LIN {X 0,Y 238.597,Z 271.892,A -85,B 0,C 180,E1 -19740.745,E2 -19740.745} C_VEL
LIN {X 0,Y 234.921,Z 263.135,A -85,B 0,C 180,E1 -19741.833,E2 -19741.833} C_VEL
LIN {X 0,Y 234.766,Z 262.386,A -85,B 0,C 180,E1 -19741.948,E2 -19741.948} C_VEL
LIN {X 0,Y 234.827,Z 259.801,A -85,B 0,C 180,E1 -19746.092,E2 -19746.092} C_VEL
LIN {X 0,Y 234.795,Z 259.401,A -85,B 0,C 180,E1 -19746.773,E2 -19746.773} C_VEL
LIN {X 0,Y 234.887,Z 259.23,A -85,B 0,C 180,E1 -19748.927,E2 -19748.927} C_VEL
LIN {X 0,Y 234.889,Z 259.225,A -85,B 0,C 180,E1 -19753.486,E2 -19753.486} C_VEL
LIN {X 0,Y 234.888,Z 259.222,A -85,B 0,C 180,E1 -19756.514,E2 -19756.514} C_VEL
LIN {X 0,Y 234.92,Z 259.222,A -85,B 0,C 180,E1 -19761.079,E2 -19761.079} C_VEL
LIN {X 0,Y 234.932,Z 259.222,A -85,B 0,C 180,E1 -19765.362,E2 -19765.362} C_VEL
LIN {X 0,Y 234.9,Z 259.224,A -85,B 0,C 180,E1 -19769.427,E2 -19769.427} C_VEL
LIN {X 0,Y 234.97,Z 259.215,A -85,B 0,C 180,E1 -19773.806,E2 -19773.806} C_VEL
LIN {X 0,Y 234.99,Z 259.212,A -85,B 0,C 180,E1 -19778.968,E2 -19778.968} C_VEL
LIN {X 0,Y 235.057,Z 259.206,A -85,B 0,C 180,E1 -19783.092,E2 -19783.092} C_VEL
LIN {X 0,Y 235.116,Z 259.196,A -85,B 0,C 180,E1 -19787.922,E2 -19787.922} C_VEL
LIN {X 0,Y 235.392,Z 259.162,A -85,B 0,C 180,E1 -19791.415,E2 -19791.415} C_VEL
LIN {X 0,Y 235.406,Z 259.16,A -85,B 0,C 180,E1 -19793.141,E2 -19793.141} C_VEL
LIN {X 0,Y 235.582,Z 259.141,A -85,B 0,C 180,E1 -19798.29,E2 -19798.29} C_VEL
LIN {X 0,Y 235.597,Z 259.138,A -85,B 0,C 180,E1 -19801.709,E2 -19801.709} C_VEL
LIN {X 0,Y 235.37,Z 259.165,A -85,B 0,C 180,E1 -19806.86,E2 -19806.86} C_VEL
LIN {X 0,Y 235.216,Z 259.185,A -85,B 0,C 180,E1 -19810.327,E2 -19810.327} C_VEL
LIN {X 0,Y 235.116,Z 259.195,A -85,B 0,C 180,E1 -19815.606,E2 -19815.606} C_VEL
LIN {X 0,Y 235.005,Z 259.212,A -85,B 0,C 180,E1 -19819.206,E2 -19819.206} C_VEL
LIN {X 0,Y 234.927,Z 259.223,A -85,B 0,C 180,E1 -19822.886,E2 -19822.886} C_VEL
LIN {X 0,Y 234.927,Z 259.226,A -85,B 0,C 180,E1 -19826.663,E2 -19826.663} C_VEL
LIN {X 0,Y 234.937,Z 259.227,A -85,B 0,C 180,E1 -19831.568,E2 -19831.568} C_VEL
LIN {X 0,Y 234.987,Z 259.521,A -85,B 0,C 180,E1 -19832.571,E2 -19832.571} C_VEL
LIN {X 0,Y 235.549,Z 262.75,A -85,B 0,C 180,E1 -19836.636,E2 -19836.636} C_VEL
LIN {X 0,Y 236.203,Z 266.509,A -85,B 0,C 180,E1 -19840.889,E2 -19840.889} C_VEL
LIN {X 0,Y 237.07,Z 270.768,A -85,B 0,C 180,E1 -19845.356,E2 -19845.356} C_VEL
LIN {X 0,Y 237.855,Z 274.98,A -85,B 0,C 180,E1 -19849.455,E2 -19849.455} C_VEL
LIN {X 0,Y 237.937,Z 275.641,A -85,B 0,C 180,E1 -19850.071,E2 -19850.071} C_VEL
LIN {X 0,Y 237.706,Z 276.681,A -85,B 0,C 180,E1 -19850.982,E2 -19850.982} C_VEL
LIN {X 0,Y 236.882,Z 277.795,A -85,B 0,C 180,E1 -19851.872,E2 -19851.872} C_VEL
LIN {X 0,Y 234.22,Z 280.117,A -85,B 0,C 180,E1 -19853.609,E2 -19853.609} C_VEL
LIN {X 0,Y 231.328,Z 282.486,A -85,B 0,C 180,E1 -19855.381,E2 -19855.381} C_VEL
LIN {X 0,Y 229.905,Z 284.219,A -85,B 0,C 180,E1 -19856.776,E2 -19856.776} C_VEL
LIN {X 0,Y 229.7,Z 284.777,A -85,B 0,C 180,E1 -19857.256,E2 -19857.256} C_VEL
LIN {X 0,Y 233.573,Z 300.662,A -85,B 0,C 180,E1 -19858.908,E2 -19858.908} C_VEL
LIN {X 0,Y 235.544,Z 312.113,A -85,B 0,C 180,E1 -19860.268,E2 -19860.268} C_VEL
LIN {X 0,Y 236.725,Z 323.693,A -85,B 0,C 180,E1 -19861.844,E2 -19861.844} C_VEL
LIN {X 0,Y 237.034,Z 334.803,A -85,B 0,C 180,E1 -19863.593,E2 -19863.593} C_VEL
LIN {X 0,Y 236.7,Z 344.769,A -85,B 0,C 180,E1 -19865.438,E2 -19865.438} C_VEL
LIN {X 0,Y 234.724,Z 352.959,A -85,B 0,C 180,E1 -19867.093,E2 -19867.093} C_VEL
LIN {X 0,Y 232.482,Z 361.592,A -85,B 0,C 180,E1 -19869.232,E2 -19869.232} C_VEL
LIN {X 0,Y 230.493,Z 369.799,A -85,B 0,C 180,E1 -19871.788,E2 -19871.788} C_VEL
LIN {X 0,Y 228.678,Z 376.512,A -85,B 0,C 180,E1 -19874.4,E2 -19874.4} C_VEL
LIN {X 0,Y 227.13,Z 382.668,A -85,B 0,C 180,E1 -19877.491,E2 -19877.491} C_VEL
LIN {X 0,Y 226.362,Z 386.685,A -85,B 0,C 180,E1 -19880.168,E2 -19880.168} C_VEL
LIN {X 0,Y 225.939,Z 389.662,A -85,B 0,C 180,E1 -19882.853,E2 -19882.853} C_VEL
LIN {X 0,Y 225.845,Z 391.153,A -85,B 0,C 180,E1 -19884.748,E2 -19884.748} C_VEL
LIN {X 0,Y 225.843,Z 392.104,A -85,B 0,C 180,E1 -19886.432,E2 -19886.432} C_VEL
LIN {X 0,Y 225.89,Z 392.728,A -85,B 0,C 180,E1 -19888.217,E2 -19888.217} C_VEL
LIN {X 0,Y 225.95,Z 392.949,A -85,B 0,C 180,E1 -19890,E2 -19890} C_VEL
LIN {X 0,Y 225.89,Z 392.72,A -85,B 0,C 180,E1 -19891.783,E2 -19891.783} C_VEL
LIN {X 0,Y 225.839,Z 392.091,A -85,B 0,C 180,E1 -19893.569,E2 -19893.569} C_VEL
LIN {X 0,Y 225.842,Z 391.068,A -85,B 0,C 180,E1 -19895.357,E2 -19895.357} C_VEL
LIN {X 0,Y 225.937,Z 389.637,A -85,B 0,C 180,E1 -19897.148,E2 -19897.148} C_VEL
LIN {X 0,Y 226.357,Z 386.646,A -85,B 0,C 180,E1 -19899.833,E2 -19899.833} C_VEL
LIN {X 0,Y 227.131,Z 382.613,A -85,B 0,C 180,E1 -19902.51,E2 -19902.51} C_VEL
LIN {X 0,Y 228.676,Z 376.437,A -85,B 0,C 180,E1 -19905.6,E2 -19905.6} C_VEL
LIN {X 0,Y 230.502,Z 369.708,A -85,B 0,C 180,E1 -19908.212,E2 -19908.212} C_VEL
LIN {X 0,Y 232.694,Z 360.843,A -85,B 0,C 180,E1 -19910.942,E2 -19910.942} C_VEL
LIN {X 0,Y 234.721,Z 352.815,A -85,B 0,C 180,E1 -19912.908,E2 -19912.908} C_VEL
LIN {X 0,Y 236.682,Z 344.6,A -85,B 0,C 180,E1 -19914.565,E2 -19914.565} C_VEL
LIN {X 0,Y 236.994,Z 334.585,A -85,B 0,C 180,E1 -19916.412,E2 -19916.412} C_VEL
LIN {X 0,Y 236.678,Z 323.434,A -85,B 0,C 180,E1 -19918.158,E2 -19918.158} C_VEL
LIN {X 0,Y 235.469,Z 311.893,A -85,B 0,C 180,E1 -19919.725,E2 -19919.725} C_VEL
LIN {X 0,Y 233.198,Z 299.127,A -85,B 0,C 180,E1 -19921.229,E2 -19921.229} C_VEL
LIN {X 0,Y 230.268,Z 287.553,A -85,B 0,C 180,E1 -19922.422,E2 -19922.422} C_VEL
LIN {X 0,Y 229.666,Z 284.769,A -85,B 0,C 180,E1 -19922.666,E2 -19922.666} C_VEL
LIN {X 0,Y 230.806,Z 280.466,A -85,B 0,C 180,E1 -19926.426,E2 -19926.426} C_VEL
LIN {X 0,Y 231.021,Z 278.054,A -85,B 0,C 180,E1 -19928.629,E2 -19928.629} C_VEL
LIN {X 0,Y 230.853,Z 276.123,A -85,B 0,C 180,E1 -19930.439,E2 -19930.439} C_VEL
LIN {X 0,Y 230.037,Z 271.961,A -85,B 0,C 180,E1 -19934.644,E2 -19934.644} C_VEL
LIN {X 0,Y 229.522,Z 269.108,A -85,B 0,C 180,E1 -19937.651,E2 -19937.651} C_VEL
LIN {X 0,Y 228.67,Z 264.453,A -85,B 0,C 180,E1 -19943.044,E2 -19943.044} C_VEL
LIN {X 0,Y 228.208,Z 261.833,A -85,B 0,C 180,E1 -19946.335,E2 -19946.335} C_VEL
LIN {X 0,Y 227.893,Z 260.097,A -85,B 0,C 180,E1 -19948.761,E2 -19948.761} C_VEL
LIN {X 0,Y 227.906,Z 260.098,A -85,B 0,C 180,E1 -19953.418,E2 -19953.418} C_VEL
LIN {X 0,Y 227.95,Z 260.093,A -85,B 0,C 180,E1 -19958.286,E2 -19958.286} C_VEL
LIN {X 0,Y 228.037,Z 260.08,A -85,B 0,C 180,E1 -19962.827,E2 -19962.827} C_VEL
LIN {X 0,Y 228.075,Z 260.076,A -85,B 0,C 180,E1 -19967.543,E2 -19967.543} C_VEL
LIN {X 0,Y 228.266,Z 260.051,A -85,B 0,C 180,E1 -19971.145,E2 -19971.145} C_VEL
LIN {X 0,Y 228.321,Z 260.043,A -85,B 0,C 180,E1 -19972.928,E2 -19972.928} C_VEL
LIN {X 0,Y 228.558,Z 260.014,A -85,B 0,C 180,E1 -19978.238,E2 -19978.238} C_VEL
LIN {X 0,Y 228.542,Z 260.018,A -85,B 0,C 180,E1 -19981.762,E2 -19981.762} C_VEL
LIN {X 0,Y 228.319,Z 260.044,A -85,B 0,C 180,E1 -19987.073,E2 -19987.073} C_VEL
LIN {X 0,Y 228.146,Z 260.066,A -85,B 0,C 180,E1 -19990.651,E2 -19990.651} C_VEL
LIN {X 0,Y 228.041,Z 260.078,A -85,B 0,C 180,E1 -19994.274,E2 -19994.274} C_VEL
LIN {X 0,Y 227.957,Z 260.086,A -85,B 0,C 180,E1 -19997.957,E2 -19997.957} C_VEL
LIN {X 0,Y 227.923,Z 260.094,A -85,B 0,C 180,E1 -20002.323,E2 -20002.323} C_VEL
LIN {X 0,Y 227.925,Z 260.094,A -85,B 0,C 180,E1 -20006.592,E2 -20006.592} C_VEL
LIN {X 0,Y 227.876,Z 260.101,A -85,B 0,C 180,E1 -20010.281,E2 -20010.281} C_VEL
LIN {X 0,Y 227.88,Z 260.098,A -85,B 0,C 180,E1 -20013.72,E2 -20013.72} C_VEL
LIN {X 0,Y 227.847,Z 260.105,A -85,B 0,C 180,E1 -20018.091,E2 -20018.091} C_VEL
LIN {X 0,Y 227.814,Z 260.106,A -85,B 0,C 180,E1 -20022.742,E2 -20022.742} C_VEL
LIN {X 0,Y 227.811,Z 260.106,A -85,B 0,C 180,E1 -20027.257,E2 -20027.257} C_VEL
LIN {X 0,Y 227.816,Z 260.107,A -85,B 0,C 180,E1 -20030.465,E2 -20030.465} C_VEL
LIN {X 0,Y 227.783,Z 260.111,A -85,B 0,C 180,E1 -20031.896,E2 -20031.896} C_VEL
LIN {X 0,Y 227.833,Z 261.048,A -85,B 0,C 180,E1 -20034.119,E2 -20034.119} C_VEL
LIN {X 0,Y 227.804,Z 262.883,A -85,B 0,C 180,E1 -20037.124,E2 -20037.124} C_VEL
LIN {X 0,Y 228.901,Z 265.947,A -85,B 0,C 180,E1 -20037.508,E2 -20037.508} C_VEL
LIN {X 0,Y 233.368,Z 276.685,A -85,B 0,C 180,E1 -20038.978,E2 -20038.978} C_VEL
LIN {X 0,Y 236.842,Z 287.16,A -85,B 0,C 180,E1 -20040.513,E2 -20040.513} C_VEL
LIN {X 0,Y 239.401,Z 297.64,A -85,B 0,C 180,E1 -20042.174,E2 -20042.174} C_VEL
LIN {X 0,Y 240.91,Z 306.572,A -85,B 0,C 180,E1 -20043.735,E2 -20043.735} C_VEL
LIN {X 0,Y 241.071,Z 308.452,A -85,B 0,C 180,E1 -20044.068,E2 -20044.068} C_VEL
LIN {X 0,Y 239.057,Z 318.286,A -85,B 0,C 180,E1 -20045.695,E2 -20045.695} C_VEL
LIN {X 0,Y 236.799,Z 328.203,A -85,B 0,C 180,E1 -20047.764,E2 -20047.764} C_VEL
LIN {X 0,Y 234.201,Z 337.802,A -85,B 0,C 180,E1 -20050.269,E2 -20050.269} C_VEL
LIN {X 0,Y 231.99,Z 345.446,A -85,B 0,C 180,E1 -20052.82,E2 -20052.82} C_VEL
LIN {X 0,Y 230.501,Z 350.658,A -85,B 0,C 180,E1 -20054.979,E2 -20054.979} C_VEL
LIN {X 0,Y 228.915,Z 355.716,A -85,B 0,C 180,E1 -20057.589,E2 -20057.589} C_VEL
LIN {X 0,Y 227.809,Z 359.633,A -85,B 0,C 180,E1 -20060.231,E2 -20060.231} C_VEL
LIN {X 0,Y 227.03,Z 362.522,A -85,B 0,C 180,E1 -20062.887,E2 -20062.887} C_VEL
LIN {X 0,Y 226.641,Z 363.904,A -85,B 0,C 180,E1 -20064.662,E2 -20064.662} C_VEL
LIN {X 0,Y 226.13,Z 365.496,A -85,B 0,C 180,E1 -20068.219,E2 -20068.219} C_VEL
LIN {X 0,Y 226.084,Z 365.723,A -85,B 0,C 180,E1 -20070,E2 -20070} C_VEL
LIN {X 0,Y 226.313,Z 364.946,A -85,B 0,C 180,E1 -20073.561,E2 -20073.561} C_VEL
LIN {X 0,Y 226.627,Z 363.983,A -85,B 0,C 180,E1 -20075.338,E2 -20075.338} C_VEL
LIN {X 0,Y 227.3,Z 361.44,A -85,B 0,C 180,E1 -20078.339,E2 -20078.339} C_VEL
LIN {X 0,Y 228.481,Z 357.329,A -85,B 0,C 180,E1 -20081.533,E2 -20081.533} C_VEL
LIN {X 0,Y 229.836,Z 352.722,A -85,B 0,C 180,E1 -20084.16,E2 -20084.16} C_VEL
LIN {X 0,Y 231.915,Z 345.77,A -85,B 0,C 180,E1 -20087.185,E2 -20087.185} C_VEL
LIN {X 0,Y 234.129,Z 338.223,A -85,B 0,C 180,E1 -20089.737,E2 -20089.737} C_VEL
LIN {X 0,Y 236.736,Z 328.716,A -85,B 0,C 180,E1 -20092.241,E2 -20092.241} C_VEL
LIN {X 0,Y 238.959,Z 318.91,A -85,B 0,C 180,E1 -20094.315,E2 -20094.315} C_VEL
LIN {X 0,Y 241.151,Z 308.24,A -85,B 0,C 180,E1 -20096.091,E2 -20096.091} C_VEL
LIN {X 0,Y 239.528,Z 298.088,A -85,B 0,C 180,E1 -20097.884,E2 -20097.884} C_VEL
LIN {X 0,Y 237.21,Z 288.374,A -85,B 0,C 180,E1 -20099.441,E2 -20099.441} C_VEL
LIN {X 0,Y 233.811,Z 277.855,A -85,B 0,C 180,E1 -20100.998,E2 -20100.998} C_VEL
LIN {X 0,Y 229.349,Z 266.623,A -85,B 0,C 180,E1 -20102.523,E2 -20102.523} C_VEL
LIN {X 0,Y 227.97,Z 263.675,A -85,B 0,C 180,E1 -20102.921,E2 -20102.921} C_VEL
LIN {X 0,Y 227.812,Z 262.875,A -85,B 0,C 180,E1 -20103.011,E2 -20103.011} C_VEL
LIN {X 0,Y 227.807,Z 260.688,A -85,B 0,C 180,E1 -20106.667,E2 -20106.667} C_VEL
LIN {X 0,Y 227.783,Z 260.115,A -85,B 0,C 180,E1 -20108.103,E2 -20108.103} C_VEL
LIN {X 0,Y 227.808,Z 260.109,A -85,B 0,C 180,E1 -20112.233,E2 -20112.233} C_VEL
LIN {X 0,Y 227.835,Z 260.105,A -85,B 0,C 180,E1 -20115.193,E2 -20115.193} C_VEL
LIN {X 0,Y 227.827,Z 260.106,A -85,B 0,C 180,E1 -20119.623,E2 -20119.623} C_VEL
LIN {X 0,Y 227.883,Z 260.1,A -85,B 0,C 180,E1 -20124.128,E2 -20124.128} C_VEL
LIN {X 0,Y 227.857,Z 260.099,A -85,B 0,C 180,E1 -20128.376,E2 -20128.376} C_VEL
LIN {X 0,Y 227.856,Z 260.101,A -85,B 0,C 180,E1 -20132.441,E2 -20132.441} C_VEL
LIN {X 0,Y 227.896,Z 260.097,A -85,B 0,C 180,E1 -20136.365,E2 -20136.365} C_VEL
LIN {X 0,Y 227.924,Z 260.093,A -85,B 0,C 180,E1 -20140.173,E2 -20140.173} C_VEL
LIN {X 0,Y 228.025,Z 260.08,A -85,B 0,C 180,E1 -20143.895,E2 -20143.895} C_VEL
LIN {X 0,Y 228.071,Z 260.075,A -85,B 0,C 180,E1 -20147.543,E2 -20147.543} C_VEL
LIN {X 0,Y 228.327,Z 260.044,A -85,B 0,C 180,E1 -20151.147,E2 -20151.147} C_VEL
LIN {X 0,Y 228.359,Z 260.037,A -85,B 0,C 180,E1 -20152.929,E2 -20152.929} C_VEL
LIN {X 0,Y 228.541,Z 260.018,A -85,B 0,C 180,E1 -20158.238,E2 -20158.238} C_VEL
LIN {X 0,Y 228.556,Z 260.015,A -85,B 0,C 180,E1 -20161.762,E2 -20161.762} C_VEL
LIN {X 0,Y 228.32,Z 260.043,A -85,B 0,C 180,E1 -20167.072,E2 -20167.072} C_VEL
LIN {X 0,Y 228.147,Z 260.067,A -85,B 0,C 180,E1 -20170.651,E2 -20170.651} C_VEL
LIN {X 0,Y 228.066,Z 260.076,A -85,B 0,C 180,E1 -20174.272,E2 -20174.272} C_VEL
LIN {X 0,Y 228.003,Z 260.083,A -85,B 0,C 180,E1 -20177.953,E2 -20177.953} C_VEL
LIN {X 0,Y 227.909,Z 260.098,A -85,B 0,C 180,E1 -20182.316,E2 -20182.316} C_VEL
LIN {X 0,Y 227.904,Z 260.102,A -85,B 0,C 180,E1 -20186.583,E2 -20186.583} C_VEL
LIN {X 0,Y 227.892,Z 260.111,A -85,B 0,C 180,E1 -20191.239,E2 -20191.239} C_VEL
LIN {X 0,Y 228.497,Z 263.553,A -85,B 0,C 180,E1 -20195.76,E2 -20195.76} C_VEL
LIN {X 0,Y 229.102,Z 267.188,A -85,B 0,C 180,E1 -20200.106,E2 -20200.106} C_VEL
LIN {X 0,Y 229.939,Z 271.349,A -85,B 0,C 180,E1 -20204.667,E2 -20204.667} C_VEL
LIN {X 0,Y 230.527,Z 274.499,A -85,B 0,C 180,E1 -20207.878,E2 -20207.878} C_VEL
LIN {X 0,Y 230.946,Z 276.956,A -85,B 0,C 180,E1 -20210.278,E2 -20210.278} C_VEL
LIN {X 0,Y 231.016,Z 279.355,A -85,B 0,C 180,E1 -20212.523,E2 -20212.523} C_VEL
LIN {X 0,Y 230.248,Z 282.743,A -85,B 0,C 180,E1 -20215.501,E2 -20215.501} C_VEL
LIN {X 0,Y 229.7,Z 284.777,A -85,B 0,C 180,E1 -20217.256,E2 -20217.256} C_VEL
LIN {X 0,Y 233.119,Z 287.593,A -85,B 0,C 180,E1 -20217.954,E2 -20217.954} C_VEL
LIN {X 0,Y 234.392,Z 290.07,A -85,B 0,C 180,E1 -20218.296,E2 -20218.296} C_VEL
LIN {X 0,Y 234.315,Z 292.249,A -85,B 0,C 180,E1 -20218.385,E2 -20218.385} C_VEL
LIN {X 0,Y 232.818,Z 294.919,A -85,B 0,C 180,E1 -20218.341,E2 -20218.341} C_VEL
LIN {X 0,Y 229.863,Z 298.76,A -85,B 0,C 180,E1 -20218.209,E2 -20218.209} C_VEL
LIN {X 0,Y 228.983,Z 301.023,A -85,B 0,C 180,E1 -20218.262,E2 -20218.262} C_VEL
LIN {X 0,Y 228.222,Z 301.846,A -85,B 0,C 180,E1 -20218.225,E2 -20218.225} C_VEL
LIN {X 0,Y 227.828,Z 304.979,A -85,B 0,C 180,E1 -20218.455,E2 -20218.455} C_VEL
LIN {X 0,Y 227.879,Z 305.401,A -85,B 0,C 180,E1 -20218.508,E2 -20218.508} C_VEL
LIN {X 0,Y 229.606,Z 317.436,A -85,B 0,C 180,E1 -20220.106,E2 -20220.106} C_VEL
LIN {X 0,Y 230.33,Z 328.16,A -85,B 0,C 180,E1 -20221.729,E2 -20221.729} C_VEL
LIN {X 0,Y 230.311,Z 338.321,A -85,B 0,C 180,E1 -20223.494,E2 -20223.494} C_VEL
LIN {X 0,Y 229.815,Z 346.502,A -85,B 0,C 180,E1 -20225.135,E2 -20225.135} C_VEL
LIN {X 0,Y 227.187,Z 356.129,A -85,B 0,C 180,E1 -20227.252,E2 -20227.252} C_VEL
LIN {X 0,Y 224.778,Z 364.945,A -85,B 0,C 180,E1 -20229.718,E2 -20229.718} C_VEL
LIN {X 0,Y 222.982,Z 371.777,A -85,B 0,C 180,E1 -20232.103,E2 -20232.103} C_VEL
LIN {X 0,Y 221.533,Z 377.087,A -85,B 0,C 180,E1 -20234.356,E2 -20234.356} C_VEL
LIN {X 0,Y 220.146,Z 382.237,A -85,B 0,C 180,E1 -20237.087,E2 -20237.087} C_VEL
LIN {X 0,Y 219.339,Z 386.256,A -85,B 0,C 180,E1 -20239.85,E2 -20239.85} C_VEL
LIN {X 0,Y 218.866,Z 389.233,A -85,B 0,C 180,E1 -20242.621,E2 -20242.621} C_VEL
LIN {X 0,Y 218.769,Z 390.865,A -85,B 0,C 180,E1 -20244.799,E2 -20244.799} C_VEL
LIN {X 0,Y 218.821,Z 392.302,A -85,B 0,C 180,E1 -20248.16,E2 -20248.16} C_VEL
LIN {X 0,Y 218.878,Z 392.523,A -85,B 0,C 180,E1 -20250,E2 -20250} C_VEL
LIN {X 0,Y 218.82,Z 392.294,A -85,B 0,C 180,E1 -20251.841,E2 -20251.841} C_VEL
LIN {X 0,Y 218.769,Z 390.848,A -85,B 0,C 180,E1 -20255.199,E2 -20255.199} C_VEL
LIN {X 0,Y 218.862,Z 389.206,A -85,B 0,C 180,E1 -20257.38,E2 -20257.38} C_VEL
LIN {X 0,Y 219.335,Z 386.216,A -85,B 0,C 180,E1 -20260.151,E2 -20260.151} C_VEL
LIN {X 0,Y 220.146,Z 382.181,A -85,B 0,C 180,E1 -20262.913,E2 -20262.913} C_VEL
LIN {X 0,Y 221.825,Z 376.007,A -85,B 0,C 180,E1 -20266.095,E2 -20266.095} C_VEL
LIN {X 0,Y 223.75,Z 369.277,A -85,B 0,C 180,E1 -20268.781,E2 -20268.781} C_VEL
LIN {X 0,Y 225.895,Z 360.927,A -85,B 0,C 180,E1 -20271.442,E2 -20271.442} C_VEL
LIN {X 0,Y 228.185,Z 352.383,A -85,B 0,C 180,E1 -20273.603,E2 -20273.603} C_VEL
LIN {X 0,Y 229.923,Z 345.243,A -85,B 0,C 180,E1 -20275.095,E2 -20275.095} C_VEL
LIN {X 0,Y 230.367,Z 334.133,A -85,B 0,C 180,E1 -20277.234,E2 -20277.234} C_VEL
LIN {X 0,Y 230.076,Z 323.178,A -85,B 0,C 180,E1 -20279.014,E2 -20279.014} C_VEL
LIN {X 0,Y 228.809,Z 311.445,A -85,B 0,C 180,E1 -20280.679,E2 -20280.679} C_VEL
LIN {X 0,Y 226.573,Z 298.834,A -85,B 0,C 180,E1 -20282.234,E2 -20282.234} C_VEL
LIN {X 0,Y 223.623,Z 287.409,A -85,B 0,C 180,E1 -20283.489,E2 -20283.489} C_VEL
LIN {X 0,Y 222.922,Z 284.281,A -85,B 0,C 180,E1 -20283.82,E2 -20283.82} C_VEL
LIN {X 0,Y 223.788,Z 281.153,A -85,B 0,C 180,E1 -20286.634,E2 -20286.634} C_VEL
LIN {X 0,Y 223.998,Z 278.82,A -85,B 0,C 180,E1 -20288.867,E2 -20288.867} C_VEL
LIN {X 0,Y 223.456,Z 275.247,A -85,B 0,C 180,E1 -20292.46,E2 -20292.46} C_VEL
LIN {X 0,Y 222.685,Z 271.445,A -85,B 0,C 180,E1 -20296.543,E2 -20296.543} C_VEL
LIN {X 0,Y 222,Z 267.817,A -85,B 0,C 180,E1 -20300.717,E2 -20300.717} C_VEL
LIN {X 0,Y 221.432,Z 264.256,A -85,B 0,C 180,E1 -20305.159,E2 -20305.159} C_VEL
LIN {X 0,Y 220.833,Z 260.977,A -85,B 0,C 180,E1 -20309.918,E2 -20309.918} C_VEL
LIN {X 0,Y 220.86,Z 260.976,A -85,B 0,C 180,E1 -20313.545,E2 -20313.545} C_VEL
LIN {X 0,Y 220.856,Z 260.977,A -85,B 0,C 180,E1 -20317.551,E2 -20317.551} C_VEL
LIN {X 0,Y 220.987,Z 260.96,A -85,B 0,C 180,E1 -20322.572,E2 -20322.572} C_VEL
LIN {X 0,Y 221.015,Z 260.954,A -85,B 0,C 180,E1 -20327.139,E2 -20327.139} C_VEL
LIN {X 0,Y 221.204,Z 260.93,A -85,B 0,C 180,E1 -20330.859,E2 -20330.859} C_VEL
LIN {X 0,Y 221.14,Z 260.939,A -85,B 0,C 180,E1 -20334.529,E2 -20334.529} C_VEL
LIN {X 0,Y 221.515,Z 260.892,A -85,B 0,C 180,E1 -20338.182,E2 -20338.182} C_VEL
LIN {X 0,Y 221.476,Z 260.898,A -85,B 0,C 180,E1 -20341.819,E2 -20341.819} C_VEL
LIN {X 0,Y 221.255,Z 260.926,A -85,B 0,C 180,E1 -20347.3,E2 -20347.3} C_VEL
LIN {X 0,Y 221.066,Z 260.949,A -85,B 0,C 180,E1 -20350.997,E2 -20350.997} C_VEL
LIN {X 0,Y 220.982,Z 260.959,A -85,B 0,C 180,E1 -20356.633,E2 -20356.633} C_VEL
LIN {X 0,Y 220.881,Z 260.97,A -85,B 0,C 180,E1 -20360.487,E2 -20360.487} C_VEL
LIN {X 0,Y 220.85,Z 260.975,A -85,B 0,C 180,E1 -20364.437,E2 -20364.437} C_VEL
LIN {X 0,Y 220.807,Z 260.98,A -85,B 0,C 180,E1 -20368.518,E2 -20368.518} C_VEL
LIN {X 0,Y 220.815,Z 260.979,A -85,B 0,C 180,E1 -20372.757,E2 -20372.757} C_VEL
LIN {X 0,Y 220.814,Z 260.979,A -85,B 0,C 180,E1 -20377.278,E2 -20377.278} C_VEL
LIN {X 0,Y 220.773,Z 260.984,A -85,B 0,C 180,E1 -20381.952,E2 -20381.952} C_VEL
LIN {X 0,Y 220.776,Z 260.983,A -85,B 0,C 180,E1 -20385.546,E2 -20385.546} C_VEL
LIN {X 0,Y 220.771,Z 260.985,A -85,B 0,C 180,E1 -20390.455,E2 -20390.455} C_VEL
LIN {X 0,Y 220.788,Z 261.541,A -85,B 0,C 180,E1 -20392.785,E2 -20392.785} C_VEL
LIN {X 0,Y 220.806,Z 263.348,A -85,B 0,C 180,E1 -20395.941,E2 -20395.941} C_VEL
LIN {X 0,Y 221.979,Z 266.534,A -85,B 0,C 180,E1 -20396.368,E2 -20396.368} C_VEL
LIN {X 0,Y 225.659,Z 274.82,A -85,B 0,C 180,E1 -20397.581,E2 -20397.581} C_VEL
LIN {X 0,Y 229.593,Z 285.875,A -85,B 0,C 180,E1 -20399.279,E2 -20399.279} C_VEL
LIN {X 0,Y 232.42,Z 296.741,A -85,B 0,C 180,E1 -20401.065,E2 -20401.065} C_VEL
LIN {X 0,Y 234.271,Z 307.231,A -85,B 0,C 180,E1 -20402.966,E2 -20402.966} C_VEL
LIN {X 0,Y 234.433,Z 310.221,A -85,B 0,C 180,E1 -20403.516,E2 -20403.516} C_VEL
LIN {X 0,Y 232.247,Z 320.254,A -85,B 0,C 180,E1 -20405.279,E2 -20405.279} C_VEL
LIN {X 0,Y 229.805,Z 330.399,A -85,B 0,C 180,E1 -20407.525,E2 -20407.525} C_VEL
LIN {X 0,Y 227.55,Z 338.231,A -85,B 0,C 180,E1 -20409.667,E2 -20409.667} C_VEL
LIN {X 0,Y 225.229,Z 345.875,A -85,B 0,C 180,E1 -20412.287,E2 -20412.287} C_VEL
LIN {X 0,Y 223.679,Z 351.086,A -85,B 0,C 180,E1 -20414.51,E2 -20414.51} C_VEL
LIN {X 0,Y 222.005,Z 356.144,A -85,B 0,C 180,E1 -20417.197,E2 -20417.197} C_VEL
LIN {X 0,Y 220.831,Z 360.061,A -85,B 0,C 180,E1 -20419.919,E2 -20419.919} C_VEL
LIN {X 0,Y 220.005,Z 362.949,A -85,B 0,C 180,E1 -20422.658,E2 -20422.658} C_VEL
LIN {X 0,Y 219.604,Z 364.33,A -85,B 0,C 180,E1 -20424.49,E2 -20424.49} C_VEL
LIN {X 0,Y 219.06,Z 365.922,A -85,B 0,C 180,E1 -20428.161,E2 -20428.161} C_VEL
LIN {X 0,Y 219.009,Z 366.149,A -85,B 0,C 180,E1 -20430,E2 -20430} C_VEL
LIN {X 0,Y 219.256,Z 365.372,A -85,B 0,C 180,E1 -20433.675,E2 -20433.675} C_VEL
LIN {X 0,Y 219.591,Z 364.408,A -85,B 0,C 180,E1 -20435.51,E2 -20435.51} C_VEL
LIN {X 0,Y 220.243,Z 362.044,A -85,B 0,C 180,E1 -20438.42,E2 -20438.42} C_VEL
LIN {X 0,Y 221.155,Z 359.027,A -85,B 0,C 180,E1 -20440.992,E2 -20440.992} C_VEL
LIN {X 0,Y 222.452,Z 354.8,A -85,B 0,C 180,E1 -20443.706,E2 -20443.706} C_VEL
LIN {X 0,Y 224.513,Z 348.39,A -85,B 0,C 180,E1 -20446.831,E2 -20446.831} C_VEL
LIN {X 0,Y 226.628,Z 341.341,A -85,B 0,C 180,E1 -20449.473,E2 -20449.473} C_VEL
LIN {X 0,Y 229.288,Z 332.544,A -85,B 0,C 180,E1 -20452.054,E2 -20452.054} C_VEL
LIN {X 0,Y 231.713,Z 322.981,A -85,B 0,C 180,E1 -20454.302,E2 -20454.302} C_VEL
LIN {X 0,Y 234.092,Z 312.234,A -85,B 0,C 180,E1 -20456.285,E2 -20456.285} C_VEL
LIN {X 0,Y 234.601,Z 309.666,A -85,B 0,C 180,E1 -20456.703,E2 -20456.703} C_VEL
LIN {X 0,Y 232.958,Z 299.028,A -85,B 0,C 180,E1 -20458.671,E2 -20458.671} C_VEL
LIN {X 0,Y 230.566,Z 289.121,A -85,B 0,C 180,E1 -20460.343,E2 -20460.343} C_VEL
LIN {X 0,Y 226.748,Z 277.565,A -85,B 0,C 180,E1 -20462.143,E2 -20462.143} C_VEL
LIN {X 0,Y 222.243,Z 266.899,A -85,B 0,C 180,E1 -20463.712,E2 -20463.712} C_VEL
LIN {X 0,Y 220.922,Z 264.041,A -85,B 0,C 180,E1 -20464.12,E2 -20464.12} C_VEL
LIN {X 0,Y 220.784,Z 263.355,A -85,B 0,C 180,E1 -20464.207,E2 -20464.207} C_VEL
LIN {X 0,Y 220.792,Z 261.587,A -85,B 0,C 180,E1 -20467.271,E2 -20467.271} C_VEL
LIN {X 0,Y 220.774,Z 260.988,A -85,B 0,C 180,E1 -20470.181,E2 -20470.181} C_VEL
LIN {X 0,Y 220.775,Z 260.984,A -85,B 0,C 180,E1 -20474.454,E2 -20474.454} C_VEL
LIN {X 0,Y 220.771,Z 260.985,A -85,B 0,C 180,E1 -20478.047,E2 -20478.047} C_VEL
LIN {X 0,Y 220.826,Z 260.978,A -85,B 0,C 180,E1 -20482.793,E2 -20482.793} C_VEL
LIN {X 0,Y 220.813,Z 260.98,A -85,B 0,C 180,E1 -20487.243,E2 -20487.243} C_VEL
LIN {X 0,Y 220.805,Z 260.979,A -85,B 0,C 180,E1 -20491.482,E2 -20491.482} C_VEL
LIN {X 0,Y 220.848,Z 260.975,A -85,B 0,C 180,E1 -20495.563,E2 -20495.563} C_VEL
LIN {X 0,Y 220.879,Z 260.973,A -85,B 0,C 180,E1 -20499.512,E2 -20499.512} C_VEL
LIN {X 0,Y 220.98,Z 260.96,A -85,B 0,C 180,E1 -20503.367,E2 -20503.367} C_VEL
LIN {X 0,Y 221.112,Z 260.94,A -85,B 0,C 180,E1 -20509.006,E2 -20509.006} C_VEL
LIN {X 0,Y 221.312,Z 260.915,A -85,B 0,C 180,E1 -20512.702,E2 -20512.702} C_VEL
LIN {X 0,Y 221.475,Z 260.898,A -85,B 0,C 180,E1 -20518.181,E2 -20518.181} C_VEL
LIN {X 0,Y 221.514,Z 260.893,A -85,B 0,C 180,E1 -20521.818,E2 -20521.818} C_VEL
LIN {X 0,Y 221.256,Z 260.923,A -85,B 0,C 180,E1 -20527.299,E2 -20527.299} C_VEL
LIN {X 0,Y 221.069,Z 260.947,A -85,B 0,C 180,E1 -20530.996,E2 -20530.996} C_VEL
LIN {X 0,Y 220.997,Z 260.954,A -85,B 0,C 180,E1 -20534.739,E2 -20534.739} C_VEL
LIN {X 0,Y 220.92,Z 260.967,A -85,B 0,C 180,E1 -20538.55,E2 -20538.55} C_VEL
LIN {X 0,Y 220.856,Z 260.977,A -85,B 0,C 180,E1 -20542.657,E2 -20542.657} C_VEL
LIN {X 0,Y 220.851,Z 260.98,A -85,B 0,C 180,E1 -20546.998,E2 -20546.998} C_VEL
LIN {X 0,Y 220.861,Z 261.089,A -85,B 0,C 180,E1 -20550.342,E2 -20550.342} C_VEL
LIN {X 0,Y 221.425,Z 264.32,A -85,B 0,C 180,E1 -20554.842,E2 -20554.842} C_VEL
LIN {X 0,Y 221.997,Z 267.879,A -85,B 0,C 180,E1 -20559.284,E2 -20559.284} C_VEL
LIN {X 0,Y 222.796,Z 271.947,A -85,B 0,C 180,E1 -20563.946,E2 -20563.946} C_VEL
LIN {X 0,Y 223.484,Z 275.321,A -85,B 0,C 180,E1 -20567.562,E2 -20567.562} C_VEL
LIN {X 0,Y 224,Z 278.88,A -85,B 0,C 180,E1 -20571.134,E2 -20571.134} C_VEL
LIN {X 0,Y 223.787,Z 281.256,A -85,B 0,C 180,E1 -20573.367,E2 -20573.367} C_VEL
LIN {X 0,Y 222.926,Z 284.374,A -85,B 0,C 180,E1 -20576.182,E2 -20576.182} C_VEL
LIN {X 0,Y 223.698,Z 287.564,A -85,B 0,C 180,E1 -20576.484,E2 -20576.484} C_VEL
LIN {X 0,Y 226.867,Z 299.952,A -85,B 0,C 180,E1 -20577.86,E2 -20577.86} C_VEL
LIN {X 0,Y 227.879,Z 305.401,A -85,B 0,C 180,E1 -20578.508,E2 -20578.508} C_VEL
LIN {X 0,Y 228.186,Z 310.915,A -85,B 0,C 180,E1 -20579.124,E2 -20579.124} C_VEL
LIN {X 0,Y 227.4,Z 316.485,A -85,B 0,C 180,E1 -20579.68,E2 -20579.68} C_VEL
LIN {X 0,Y 224.408,Z 328.864,A -85,B 0,C 180,E1 -20581.09,E2 -20581.09} C_VEL
LIN {X 0,Y 223.819,Z 333.8,A -85,B 0,C 180,E1 -20581.88,E2 -20581.88} C_VEL
LIN {X 0,Y 223.39,Z 343.889,A -85,B 0,C 180,E1 -20583.868,E2 -20583.868} C_VEL
LIN {X 0,Y 222.799,Z 348.194,A -85,B 0,C 180,E1 -20584.796,E2 -20584.796} C_VEL
LIN {X 0,Y 220.143,Z 357.383,A -85,B 0,C 180,E1 -20586.979,E2 -20586.979} C_VEL
LIN {X 0,Y 217.635,Z 366.311,A -85,B 0,C 180,E1 -20589.668,E2 -20589.668} C_VEL
LIN {X 0,Y 215.568,Z 373.604,A -85,B 0,C 180,E1 -20592.448,E2 -20592.448} C_VEL
LIN {X 0,Y 213.629,Z 380.203,A -85,B 0,C 180,E1 -20595.716,E2 -20595.716} C_VEL
LIN {X 0,Y 212.57,Z 384.587,A -85,B 0,C 180,E1 -20598.558,E2 -20598.558} C_VEL
LIN {X 0,Y 212.122,Z 386.916,A -85,B 0,C 180,E1 -20600.465,E2 -20600.465} C_VEL
LIN {X 0,Y 211.818,Z 388.806,A -85,B 0,C 180,E1 -20602.374,E2 -20602.374} C_VEL
LIN {X 0,Y 211.682,Z 390.597,A -85,B 0,C 180,E1 -20604.888,E2 -20604.888} C_VEL
LIN {X 0,Y 211.751,Z 391.876,A -85,B 0,C 180,E1 -20608.098,E2 -20608.098} C_VEL
LIN {X 0,Y 211.808,Z 392.097,A -85,B 0,C 180,E1 -20610,E2 -20610} C_VEL
LIN {X 0,Y 211.75,Z 391.867,A -85,B 0,C 180,E1 -20611.902,E2 -20611.902} C_VEL
LIN {X 0,Y 211.688,Z 390.569,A -85,B 0,C 180,E1 -20615.127,E2 -20615.127} C_VEL
LIN {X 0,Y 211.814,Z 388.778,A -85,B 0,C 180,E1 -20617.627,E2 -20617.627} C_VEL
LIN {X 0,Y 212.333,Z 385.787,A -85,B 0,C 180,E1 -20620.489,E2 -20620.489} C_VEL
LIN {X 0,Y 213.18,Z 381.749,A -85,B 0,C 180,E1 -20623.343,E2 -20623.343} C_VEL
LIN {X 0,Y 214.986,Z 375.576,A -85,B 0,C 180,E1 -20626.622,E2 -20626.622} C_VEL
LIN {X 0,Y 216.991,Z 368.894,A -85,B 0,C 180,E1 -20629.37,E2 -20629.37} C_VEL
LIN {X 0,Y 219.231,Z 360.493,A -85,B 0,C 180,E1 -20632.128,E2 -20632.128} C_VEL
LIN {X 0,Y 221.689,Z 351.952,A -85,B 0,C 180,E1 -20634.339,E2 -20634.339} C_VEL
LIN {X 0,Y 223.197,Z 345.885,A -85,B 0,C 180,E1 -20635.656,E2 -20635.656} C_VEL
LIN {X 0,Y 223.779,Z 334.6,A -85,B 0,C 180,E1 -20637.934,E2 -20637.934} C_VEL
LIN {X 0,Y 223.49,Z 322.761,A -85,B 0,C 180,E1 -20639.948,E2 -20639.948} C_VEL
LIN {X 0,Y 222.12,Z 310.18,A -85,B 0,C 180,E1 -20641.8,E2 -20641.8} C_VEL
LIN {X 0,Y 219.724,Z 297.178,A -85,B 0,C 180,E1 -20643.47,E2 -20643.47} C_VEL
LIN {X 0,Y 216.285,Z 284.364,A -85,B 0,C 180,E1 -20644.923,E2 -20644.923} C_VEL
LIN {X 0,Y 216.252,Z 283.776,A -85,B 0,C 180,E1 -20645.028,E2 -20645.028} C_VEL
LIN {X 0,Y 216.771,Z 281.856,A -85,B 0,C 180,E1 -20646.856,E2 -20646.856} C_VEL
LIN {X 0,Y 216.981,Z 279.706,A -85,B 0,C 180,E1 -20648.981,E2 -20648.981} C_VEL
LIN {X 0,Y 216.359,Z 275.872,A -85,B 0,C 180,E1 -20653.012,E2 -20653.012} C_VEL
LIN {X 0,Y 215.65,Z 272.478,A -85,B 0,C 180,E1 -20656.812,E2 -20656.812} C_VEL
LIN {X 0,Y 214.906,Z 268.495,A -85,B 0,C 180,E1 -20661.585,E2 -20661.585} C_VEL
LIN {X 0,Y 214.348,Z 265.055,A -85,B 0,C 180,E1 -20666.124,E2 -20666.124} C_VEL
LIN {X 0,Y 213.795,Z 261.854,A -85,B 0,C 180,E1 -20670.996,E2 -20670.996} C_VEL
LIN {X 0,Y 213.755,Z 261.861,A -85,B 0,C 180,E1 -20674.696,E2 -20674.696} C_VEL
LIN {X 0,Y 213.8,Z 261.856,A -85,B 0,C 180,E1 -20678.802,E2 -20678.802} C_VEL
LIN {X 0,Y 213.947,Z 261.836,A -85,B 0,C 180,E1 -20682.804,E2 -20682.804} C_VEL
LIN {X 0,Y 213.956,Z 261.834,A -85,B 0,C 180,E1 -20686.707,E2 -20686.707} C_VEL
LIN {X 0,Y 214.142,Z 261.81,A -85,B 0,C 180,E1 -20690.555,E2 -20690.555} C_VEL
LIN {X 0,Y 214.101,Z 261.816,A -85,B 0,C 180,E1 -20694.349,E2 -20694.349} C_VEL
LIN {X 0,Y 214.449,Z 261.772,A -85,B 0,C 180,E1 -20698.122,E2 -20698.122} C_VEL
LIN {X 0,Y 214.516,Z 261.762,A -85,B 0,C 180,E1 -20700,E2 -20700} C_VEL
LIN {X 0,Y 214.413,Z 261.777,A -85,B 0,C 180,E1 -20701.878,E2 -20701.878} C_VEL
LIN {X 0,Y 214.196,Z 261.805,A -85,B 0,C 180,E1 -20707.542,E2 -20707.542} C_VEL
LIN {X 0,Y 213.997,Z 261.827,A -85,B 0,C 180,E1 -20711.365,E2 -20711.365} C_VEL
LIN {X 0,Y 213.906,Z 261.839,A -85,B 0,C 180,E1 -20715.239,E2 -20715.239} C_VEL
LIN {X 0,Y 213.818,Z 261.852,A -85,B 0,C 180,E1 -20719.19,E2 -20719.19} C_VEL
LIN {X 0,Y 213.806,Z 261.851,A -85,B 0,C 180,E1 -20723.232,E2 -20723.232} C_VEL
LIN {X 0,Y 213.79,Z 261.854,A -85,B 0,C 180,E1 -20727.428,E2 -20727.428} C_VEL
LIN {X 0,Y 213.761,Z 261.857,A -85,B 0,C 180,E1 -20731.739,E2 -20731.739} C_VEL
LIN {X 0,Y 213.747,Z 261.855,A -85,B 0,C 180,E1 -20736.288,E2 -20736.288} C_VEL
LIN {X 0,Y 213.715,Z 261.864,A -85,B 0,C 180,E1 -20741.125,E2 -20741.125} C_VEL
LIN {X 0,Y 213.709,Z 261.865,A -85,B 0,C 180,E1 -20743.678,E2 -20743.678} C_VEL
LIN {X 0,Y 213.708,Z 261.865,A -85,B 0,C 180,E1 -20746.344,E2 -20746.344} C_VEL
LIN {X 0,Y 213.709,Z 261.865,A -85,B 0,C 180,E1 -20749.146,E2 -20749.146} C_VEL
LIN {X 0,Y 213.692,Z 262.027,A -85,B 0,C 180,E1 -20751.326,E2 -20751.326} C_VEL
LIN {X 0,Y 213.796,Z 263.927,A -85,B 0,C 180,E1 -20754.695,E2 -20754.695} C_VEL
LIN {X 0,Y 215.059,Z 267.126,A -85,B 0,C 180,E1 -20755.136,E2 -20755.136} C_VEL
LIN {X 0,Y 218.812,Z 275.077,A -85,B 0,C 180,E1 -20756.414,E2 -20756.414} C_VEL
LIN {X 0,Y 222.474,Z 285.14,A -85,B 0,C 180,E1 -20758.037,E2 -20758.037} C_VEL
LIN {X 0,Y 225.328,Z 295.285,A -85,B 0,C 180,E1 -20759.776,E2 -20759.776} C_VEL
LIN {X 0,Y 227.47,Z 306.452,A -85,B 0,C 180,E1 -20761.865,E2 -20761.865} C_VEL
LIN {X 0,Y 227.984,Z 310.661,A -85,B 0,C 180,E1 -20762.706,E2 -20762.706} C_VEL
LIN {X 0,Y 225.78,Z 320.914,A -85,B 0,C 180,E1 -20764.574,E2 -20764.574} C_VEL
LIN {X 0,Y 223.29,Z 330.828,A -85,B 0,C 180,E1 -20766.831,E2 -20766.831} C_VEL
LIN {X 0,Y 220.928,Z 338.659,A -85,B 0,C 180,E1 -20769.03,E2 -20769.03} C_VEL
LIN {X 0,Y 218.493,Z 346.304,A -85,B 0,C 180,E1 -20771.722,E2 -20771.722} C_VEL
LIN {X 0,Y 216.871,Z 351.514,A -85,B 0,C 180,E1 -20774.011,E2 -20774.011} C_VEL
LIN {X 0,Y 215.094,Z 356.573,A -85,B 0,C 180,E1 -20776.778,E2 -20776.778} C_VEL
LIN {X 0,Y 213.853,Z 360.489,A -85,B 0,C 180,E1 -20779.586,E2 -20779.586} C_VEL
LIN {X 0,Y 212.984,Z 363.376,A -85,B 0,C 180,E1 -20782.415,E2 -20782.415} C_VEL
LIN {X 0,Y 212.571,Z 364.756,A -85,B 0,C 180,E1 -20784.307,E2 -20784.307} C_VEL
LIN {X 0,Y 211.991,Z 366.348,A -85,B 0,C 180,E1 -20788.1,E2 -20788.1} C_VEL
LIN {X 0,Y 211.935,Z 366.575,A -85,B 0,C 180,E1 -20790,E2 -20790} C_VEL
LIN {X 0,Y 212.202,Z 365.797,A -85,B 0,C 180,E1 -20793.798,E2 -20793.798} C_VEL
LIN {X 0,Y 212.557,Z 364.833,A -85,B 0,C 180,E1 -20795.692,E2 -20795.692} C_VEL
LIN {X 0,Y 213.199,Z 362.626,A -85,B 0,C 180,E1 -20798.53,E2 -20798.53} C_VEL
LIN {X 0,Y 214.209,Z 359.452,A -85,B 0,C 180,E1 -20801.353,E2 -20801.353} C_VEL
LIN {X 0,Y 215.559,Z 355.226,A -85,B 0,C 180,E1 -20804.154,E2 -20804.154} C_VEL
LIN {X 0,Y 217.746,Z 348.814,A -85,B 0,C 180,E1 -20807.371,E2 -20807.371} C_VEL
LIN {X 0,Y 219.966,Z 341.765,A -85,B 0,C 180,E1 -20810.088,E2 -20810.088} C_VEL
LIN {X 0,Y 222.751,Z 332.967,A -85,B 0,C 180,E1 -20812.737,E2 -20812.737} C_VEL
LIN {X 0,Y 225.183,Z 323.786,A -85,B 0,C 180,E1 -20814.96,E2 -20814.96} C_VEL
LIN {X 0,Y 227.481,Z 313.939,A -85,B 0,C 180,E1 -20816.862,E2 -20816.862} C_VEL
LIN {X 0,Y 228.05,Z 311.372,A -85,B 0,C 180,E1 -20817.285,E2 -20817.285} C_VEL
LIN {X 0,Y 226.619,Z 301.193,A -85,B 0,C 180,E1 -20819.283,E2 -20819.283} C_VEL
LIN {X 0,Y 224.169,Z 290.62,A -85,B 0,C 180,E1 -20821.177,E2 -20821.177} C_VEL
LIN {X 0,Y 220.163,Z 278.595,A -85,B 0,C 180,E1 -20823.175,E2 -20823.175} C_VEL
LIN {X 0,Y 216.062,Z 269.052,A -85,B 0,C 180,E1 -20824.705,E2 -20824.705} C_VEL
LIN {X 0,Y 213.935,Z 264.572,A -85,B 0,C 180,E1 -20825.395,E2 -20825.395} C_VEL
LIN {X 0,Y 213.759,Z 263.827,A -85,B 0,C 180,E1 -20825.526,E2 -20825.526} C_VEL
LIN {X 0,Y 213.696,Z 262.126,A -85,B 0,C 180,E1 -20828.673,E2 -20828.673} C_VEL
LIN {X 0,Y 213.705,Z 261.865,A -85,B 0,C 180,E1 -20831.127,E2 -20831.127} C_VEL
LIN {X 0,Y 213.706,Z 261.862,A -85,B 0,C 180,E1 -20833.679,E2 -20833.679} C_VEL
LIN {X 0,Y 213.707,Z 261.86,A -85,B 0,C 180,E1 -20836.344,E2 -20836.344} C_VEL
LIN {X 0,Y 213.718,Z 261.863,A -85,B 0,C 180,E1 -20839.143,E2 -20839.143} C_VEL
LIN {X 0,Y 213.745,Z 261.859,A -85,B 0,C 180,E1 -20843.712,E2 -20843.712} C_VEL
LIN {X 0,Y 213.76,Z 261.855,A -85,B 0,C 180,E1 -20848.261,E2 -20848.261} C_VEL
LIN {X 0,Y 213.79,Z 261.853,A -85,B 0,C 180,E1 -20852.598,E2 -20852.598} C_VEL
LIN {X 0,Y 213.812,Z 261.853,A -85,B 0,C 180,E1 -20856.979,E2 -20856.979} C_VEL
LIN {X 0,Y 213.888,Z 261.839,A -85,B 0,C 180,E1 -20862.344,E2 -20862.344} C_VEL
LIN {X 0,Y 213.945,Z 261.834,A -85,B 0,C 180,E1 -20866.706,E2 -20866.706} C_VEL
LIN {X 0,Y 214.199,Z 261.803,A -85,B 0,C 180,E1 -20870.558,E2 -20870.558} C_VEL
LIN {X 0,Y 214.25,Z 261.795,A -85,B 0,C 180,E1 -20872.46,E2 -20872.46} C_VEL
LIN {X 0,Y 214.412,Z 261.777,A -85,B 0,C 180,E1 -20878.122,E2 -20878.122} C_VEL
LIN {X 0,Y 214.515,Z 261.761,A -85,B 0,C 180,E1 -20880,E2 -20880} C_VEL
LIN {X 0,Y 214.447,Z 261.773,A -85,B 0,C 180,E1 -20881.878,E2 -20881.878} C_VEL
LIN {X 0,Y 214.196,Z 261.803,A -85,B 0,C 180,E1 -20887.541,E2 -20887.541} C_VEL
LIN {X 0,Y 214.001,Z 261.828,A -85,B 0,C 180,E1 -20891.364,E2 -20891.364} C_VEL
LIN {X 0,Y 213.935,Z 261.833,A -85,B 0,C 180,E1 -20895.237,E2 -20895.237} C_VEL
LIN {X 0,Y 213.835,Z 261.849,A -85,B 0,C 180,E1 -20899.188,E2 -20899.188} C_VEL
LIN {X 0,Y 213.792,Z 261.857,A -85,B 0,C 180,E1 -20903.233,E2 -20903.233} C_VEL
LIN {X 0,Y 213.767,Z 261.864,A -85,B 0,C 180,E1 -20908.47,E2 -20908.47} C_VEL
LIN {X 0,Y 213.851,Z 262.159,A -85,B 0,C 180,E1 -20909.535,E2 -20909.535} C_VEL
LIN {X 0,Y 214.493,Z 265.936,A -85,B 0,C 180,E1 -20915.001,E2 -20915.001} C_VEL
LIN {X 0,Y 215.316,Z 270.456,A -85,B 0,C 180,E1 -20920.754,E2 -20920.754} C_VEL
LIN {X 0,Y 216.158,Z 274.73,A -85,B 0,C 180,E1 -20925.667,E2 -20925.667} C_VEL
LIN {X 0,Y 216.805,Z 278.382,A -85,B 0,C 180,E1 -20929.585,E2 -20929.585} C_VEL
LIN {X 0,Y 216.882,Z 280.78,A -85,B 0,C 180,E1 -20931.998,E2 -20931.998} C_VEL
LIN {X 0,Y 216.256,Z 283.899,A -85,B 0,C 180,E1 -20934.975,E2 -20934.975} C_VEL
LIN {X 0,Y 217.088,Z 287.342,A -85,B 0,C 180,E1 -20935.335,E2 -20935.335} C_VEL
LIN {X 0,Y 220.365,Z 300.086,A -85,B 0,C 180,E1 -20936.843,E2 -20936.843} C_VEL
LIN {X 0,Y 222.522,Z 312.758,A -85,B 0,C 180,E1 -20938.512,E2 -20938.512} C_VEL
LIN {X 0,Y 223.659,Z 325.102,A -85,B 0,C 180,E1 -20940.388,E2 -20940.388} C_VEL
LIN {X 0,Y 223.819,Z 333.8,A -85,B 0,C 180,E1 -20941.88,E2 -20941.88} C_VEL
LIN {X 0,Y 222.983,Z 338.686,A -85,B 0,C 180,E1 -20942.705,E2 -20942.705} C_VEL
LIN {X 0,Y 221.014,Z 343.43,A -85,B 0,C 180,E1 -20943.487,E2 -20943.487} C_VEL
LIN {X 0,Y 215.862,Z 352.386,A -85,B 0,C 180,E1 -20945.143,E2 -20945.143} C_VEL
LIN {X 0,Y 213.759,Z 356.62,A -85,B 0,C 180,E1 -20946.143,E2 -20946.143} C_VEL
LIN {X 0,Y 213.273,Z 357.978,A -85,B 0,C 180,E1 -20946.513,E2 -20946.513} C_VEL
LIN {X 0,Y 210.762,Z 366.532,A -85,B 0,C 180,E1 -20949.216,E2 -20949.216} C_VEL
LIN {X 0,Y 208.737,Z 373.174,A -85,B 0,C 180,E1 -20951.854,E2 -20951.854} C_VEL
LIN {X 0,Y 207.234,Z 378.066,A -85,B 0,C 180,E1 -20954.258,E2 -20954.258} C_VEL
LIN {X 0,Y 205.895,Z 382.831,A -85,B 0,C 180,E1 -20957.181,E2 -20957.181} C_VEL
LIN {X 0,Y 205.099,Z 386.488,A -85,B 0,C 180,E1 -20960.135,E2 -20960.135} C_VEL
LIN {X 0,Y 204.747,Z 388.377,A -85,B 0,C 180,E1 -20962.109,E2 -20962.109} C_VEL
LIN {X 0,Y 204.585,Z 390.35,A -85,B 0,C 180,E1 -20965.019,E2 -20965.019} C_VEL
LIN {X 0,Y 204.659,Z 391.449,A -85,B 0,C 180,E1 -20968.032,E2 -20968.032} C_VEL
LIN {X 0,Y 204.739,Z 391.671,A -85,B 0,C 180,E1 -20970,E2 -20970} C_VEL
LIN {X 0,Y 204.658,Z 391.44,A -85,B 0,C 180,E1 -20971.968,E2 -20971.968} C_VEL
LIN {X 0,Y 204.586,Z 390.329,A -85,B 0,C 180,E1 -20974.982,E2 -20974.982} C_VEL
LIN {X 0,Y 204.741,Z 388.347,A -85,B 0,C 180,E1 -20977.892,E2 -20977.892} C_VEL
LIN {X 0,Y 205.302,Z 385.355,A -85,B 0,C 180,E1 -20980.853,E2 -20980.853} C_VEL
LIN {X 0,Y 206.235,Z 381.318,A -85,B 0,C 180,E1 -20983.801,E2 -20983.801} C_VEL
LIN {X 0,Y 208.153,Z 375.144,A -85,B 0,C 180,E1 -20987.184,E2 -20987.184} C_VEL
LIN {X 0,Y 210.394,Z 367.927,A -85,B 0,C 180,E1 -20990.221,E2 -20990.221} C_VEL
LIN {X 0,Y 212.611,Z 360.057,A -85,B 0,C 180,E1 -20992.856,E2 -20992.856} C_VEL
LIN {X 0,Y 215.209,Z 351.519,A -85,B 0,C 180,E1 -20995.122,E2 -20995.122} C_VEL
LIN {X 0,Y 216.487,Z 346.527,A -85,B 0,C 180,E1 -20996.252,E2 -20996.252} C_VEL
LIN {X 0,Y 217.193,Z 335.338,A -85,B 0,C 180,E1 -20998.62,E2 -20998.62} C_VEL
LIN {X 0,Y 217.028,Z 324.042,A -85,B 0,C 180,E1 -21000.666,E2 -21000.666} C_VEL
LIN {X 0,Y 215.854,Z 311.694,A -85,B 0,C 180,E1 -21002.599,E2 -21002.599} C_VEL
LIN {X 0,Y 213.558,Z 298.913,A -85,B 0,C 180,E1 -21004.368,E2 -21004.368} C_VEL
LIN {X 0,Y 210.442,Z 286.886,A -85,B 0,C 180,E1 -21005.867,E2 -21005.867} C_VEL
LIN {X 0,Y 209.538,Z 283.555,A -85,B 0,C 180,E1 -21006.236,E2 -21006.236} C_VEL
LIN {X 0,Y 209.885,Z 281.39,A -85,B 0,C 180,E1 -21008.278,E2 -21008.278} C_VEL
LIN {X 0,Y 209.731,Z 278.996,A -85,B 0,C 180,E1 -21010.801,E2 -21010.801} C_VEL
LIN {X 0,Y 208.967,Z 275.203,A -85,B 0,C 180,E1 -21015.067,E2 -21015.067} C_VEL
LIN {X 0,Y 208.133,Z 271.076,A -85,B 0,C 180,E1 -21020.091,E2 -21020.091} C_VEL
LIN {X 0,Y 207.584,Z 267.437,A -85,B 0,C 180,E1 -21024.862,E2 -21024.862} C_VEL
LIN {X 0,Y 207.017,Z 264.37,A -85,B 0,C 180,E1 -21029.387,E2 -21029.387} C_VEL
LIN {X 0,Y 206.746,Z 262.734,A -85,B 0,C 180,E1 -21032.109,E2 -21032.109} C_VEL
LIN {X 0,Y 206.732,Z 262.737,A -85,B 0,C 180,E1 -21036.62,E2 -21036.62} C_VEL
LIN {X 0,Y 206.876,Z 262.717,A -85,B 0,C 180,E1 -21042.197,E2 -21042.197} C_VEL
LIN {X 0,Y 206.899,Z 262.713,A -85,B 0,C 180,E1 -21046.245,E2 -21046.245} C_VEL
LIN {X 0,Y 207.103,Z 262.687,A -85,B 0,C 180,E1 -21050.231,E2 -21050.231} C_VEL
LIN {X 0,Y 207.062,Z 262.693,A -85,B 0,C 180,E1 -21054.156,E2 -21054.156} C_VEL
LIN {X 0,Y 207.385,Z 262.652,A -85,B 0,C 180,E1 -21058.058,E2 -21058.058} C_VEL
LIN {X 0,Y 207.484,Z 262.638,A -85,B 0,C 180,E1 -21060,E2 -21060} C_VEL
LIN {X 0,Y 207.353,Z 262.656,A -85,B 0,C 180,E1 -21061.942,E2 -21061.942} C_VEL
LIN {X 0,Y 207.139,Z 262.683,A -85,B 0,C 180,E1 -21067.8,E2 -21067.8} C_VEL
LIN {X 0,Y 206.92,Z 262.707,A -85,B 0,C 180,E1 -21071.759,E2 -21071.759} C_VEL
LIN {X 0,Y 206.834,Z 262.72,A -85,B 0,C 180,E1 -21075.773,E2 -21075.773} C_VEL
LIN {X 0,Y 206.753,Z 262.73,A -85,B 0,C 180,E1 -21079.872,E2 -21079.872} C_VEL
LIN {X 0,Y 206.741,Z 262.731,A -85,B 0,C 180,E1 -21084.075,E2 -21084.075} C_VEL
LIN {X 0,Y 206.691,Z 262.738,A -85,B 0,C 180,E1 -21088.427,E2 -21088.427} C_VEL
LIN {X 0,Y 206.698,Z 262.737,A -85,B 0,C 180,E1 -21092.958,E2 -21092.958} C_VEL
LIN {X 0,Y 206.684,Z 262.74,A -85,B 0,C 180,E1 -21097.739,E2 -21097.739} C_VEL
LIN {X 0,Y 206.645,Z 262.746,A -85,B 0,C 180,E1 -21101.563,E2 -21101.563} C_VEL
LIN {X 0,Y 206.636,Z 262.744,A -85,B 0,C 180,E1 -21105.582,E2 -21105.582} C_VEL
LIN {X 0,Y 206.624,Z 262.748,A -85,B 0,C 180,E1 -21109.739,E2 -21109.739} C_VEL
LIN {X 0,Y 206.777,Z 264.335,A -85,B 0,C 180,E1 -21113.269,E2 -21113.269} C_VEL
LIN {X 0,Y 208.028,Z 267.569,A -85,B 0,C 180,E1 -21113.769,E2 -21113.769} C_VEL
LIN {X 0,Y 211.969,Z 275.549,A -85,B 0,C 180,E1 -21115.173,E2 -21115.173} C_VEL
LIN {X 0,Y 215.855,Z 285.932,A -85,B 0,C 180,E1 -21116.97,E2 -21116.97} C_VEL
LIN {X 0,Y 218.838,Z 296.348,A -85,B 0,C 180,E1 -21118.87,E2 -21118.87} C_VEL
LIN {X 0,Y 220.674,Z 305.734,A -85,B 0,C 180,E1 -21120.696,E2 -21120.696} C_VEL
LIN {X 0,Y 221.484,Z 312.37,A -85,B 0,C 180,E1 -21122.092,E2 -21122.092} C_VEL
LIN {X 0,Y 218.878,Z 323.523,A -85,B 0,C 180,E1 -21124.238,E2 -21124.238} C_VEL
LIN {X 0,Y 216.297,Z 332.939,A -85,B 0,C 180,E1 -21126.544,E2 -21126.544} C_VEL
LIN {X 0,Y 213.402,Z 341.811,A -85,B 0,C 180,E1 -21129.266,E2 -21129.266} C_VEL
LIN {X 0,Y 211.077,Z 348.937,A -85,B 0,C 180,E1 -21132.062,E2 -21132.062} C_VEL
LIN {X 0,Y 209.35,Z 353.743,A -85,B 0,C 180,E1 -21134.421,E2 -21134.421} C_VEL
LIN {X 0,Y 207.711,Z 358.407,A -85,B 0,C 180,E1 -21137.295,E2 -21137.295} C_VEL
LIN {X 0,Y 206.555,Z 361.966,A -85,B 0,C 180,E1 -21140.205,E2 -21140.205} C_VEL
LIN {X 0,Y 205.955,Z 363.804,A -85,B 0,C 180,E1 -21142.155,E2 -21142.155} C_VEL
LIN {X 0,Y 205.54,Z 365.182,A -85,B 0,C 180,E1 -21144.112,E2 -21144.112} C_VEL
LIN {X 0,Y 204.925,Z 366.774,A -85,B 0,C 180,E1 -21148.034,E2 -21148.034} C_VEL
LIN {X 0,Y 204.863,Z 367.001,A -85,B 0,C 180,E1 -21150,E2 -21150} C_VEL
LIN {X 0,Y 205.151,Z 366.222,A -85,B 0,C 180,E1 -21153.928,E2 -21153.928} C_VEL
LIN {X 0,Y 205.527,Z 365.258,A -85,B 0,C 180,E1 -21155.888,E2 -21155.888} C_VEL
LIN {X 0,Y 206.132,Z 363.249,A -85,B 0,C 180,E1 -21158.602,E2 -21158.602} C_VEL
LIN {X 0,Y 207.25,Z 359.879,A -85,B 0,C 180,E1 -21161.739,E2 -21161.739} C_VEL
LIN {X 0,Y 208.691,Z 355.652,A -85,B 0,C 180,E1 -21164.63,E2 -21164.63} C_VEL
LIN {X 0,Y 210.995,Z 349.239,A -85,B 0,C 180,E1 -21167.945,E2 -21167.945} C_VEL
LIN {X 0,Y 213.309,Z 342.19,A -85,B 0,C 180,E1 -21170.743,E2 -21170.743} C_VEL
LIN {X 0,Y 216.249,Z 333.389,A -85,B 0,C 180,E1 -21173.461,E2 -21173.461} C_VEL
LIN {X 0,Y 218.687,Z 324.575,A -85,B 0,C 180,E1 -21175.658,E2 -21175.658} C_VEL
LIN {X 0,Y 221.196,Z 314.361,A -85,B 0,C 180,E1 -21177.689,E2 -21177.689} C_VEL
LIN {X 0,Y 221.482,Z 311.814,A -85,B 0,C 180,E1 -21178.165,E2 -21178.165} C_VEL
LIN {X 0,Y 220.069,Z 302.115,A -85,B 0,C 180,E1 -21180.163,E2 -21180.163} C_VEL
LIN {X 0,Y 217.451,Z 290.937,A -85,B 0,C 180,E1 -21182.274,E2 -21182.274} C_VEL
LIN {X 0,Y 213.513,Z 279.329,A -85,B 0,C 180,E1 -21184.325,E2 -21184.325} C_VEL
LIN {X 0,Y 209.554,Z 270.534,A -85,B 0,C 180,E1 -21185.873,E2 -21185.873} C_VEL
LIN {X 0,Y 208.022,Z 267.566,A -85,B 0,C 180,E1 -21186.39,E2 -21186.39} C_VEL
LIN {X 0,Y 206.756,Z 264.343,A -85,B 0,C 180,E1 -21186.884,E2 -21186.884} C_VEL
LIN {X 0,Y 206.621,Z 262.751,A -85,B 0,C 180,E1 -21190.261,E2 -21190.261} C_VEL
LIN {X 0,Y 206.634,Z 262.744,A -85,B 0,C 180,E1 -21194.418,E2 -21194.418} C_VEL
LIN {X 0,Y 206.643,Z 262.745,A -85,B 0,C 180,E1 -21198.437,E2 -21198.437} C_VEL
LIN {X 0,Y 206.682,Z 262.741,A -85,B 0,C 180,E1 -21202.26,E2 -21202.26} C_VEL
LIN {X 0,Y 206.696,Z 262.738,A -85,B 0,C 180,E1 -21207.042,E2 -21207.042} C_VEL
LIN {X 0,Y 206.711,Z 262.735,A -85,B 0,C 180,E1 -21212.126,E2 -21212.126} C_VEL
LIN {X 0,Y 206.746,Z 262.732,A -85,B 0,C 180,E1 -21216.61,E2 -21216.61} C_VEL
LIN {X 0,Y 206.827,Z 262.718,A -85,B 0,C 180,E1 -21222.192,E2 -21222.192} C_VEL
LIN {X 0,Y 206.884,Z 262.712,A -85,B 0,C 180,E1 -21226.243,E2 -21226.243} C_VEL
LIN {X 0,Y 207.135,Z 262.682,A -85,B 0,C 180,E1 -21230.233,E2 -21230.233} C_VEL
LIN {X 0,Y 207.19,Z 262.675,A -85,B 0,C 180,E1 -21232.202,E2 -21232.202} C_VEL
LIN {X 0,Y 207.352,Z 262.656,A -85,B 0,C 180,E1 -21238.058,E2 -21238.058} C_VEL
LIN {X 0,Y 207.483,Z 262.637,A -85,B 0,C 180,E1 -21240,E2 -21240} C_VEL
LIN {X 0,Y 207.383,Z 262.653,A -85,B 0,C 180,E1 -21241.942,E2 -21241.942} C_VEL
LIN {X 0,Y 207.139,Z 262.683,A -85,B 0,C 180,E1 -21247.8,E2 -21247.8} C_VEL
LIN {X 0,Y 206.926,Z 262.709,A -85,B 0,C 180,E1 -21251.758,E2 -21251.758} C_VEL
LIN {X 0,Y 206.868,Z 262.714,A -85,B 0,C 180,E1 -21255.771,E2 -21255.771} C_VEL
LIN {X 0,Y 206.761,Z 262.729,A -85,B 0,C 180,E1 -21259.871,E2 -21259.871} C_VEL
LIN {X 0,Y 206.725,Z 262.738,A -85,B 0,C 180,E1 -21264.077,E2 -21264.077} C_VEL
LIN {X 0,Y 206.748,Z 262.844,A -85,B 0,C 180,E1 -21268.054,E2 -21268.054} C_VEL
LIN {X 0,Y 207.235,Z 265.929,A -85,B 0,C 180,E1 -21272.862,E2 -21272.862} C_VEL
LIN {X 0,Y 207.608,Z 267.908,A -85,B 0,C 180,E1 -21275.664,E2 -21275.664} C_VEL
LIN {X 0,Y 208.155,Z 271.128,A -85,B 0,C 180,E1 -21279.904,E2 -21279.904} C_VEL
LIN {X 0,Y 209.063,Z 275.413,A -85,B 0,C 180,E1 -21285.094,E2 -21285.094} C_VEL
LIN {X 0,Y 209.737,Z 279.074,A -85,B 0,C 180,E1 -21289.201,E2 -21289.201} C_VEL
LIN {X 0,Y 209.861,Z 281.462,A -85,B 0,C 180,E1 -21291.717,E2 -21291.717} C_VEL
LIN {X 0,Y 209.556,Z 283.43,A -85,B 0,C 180,E1 -21293.68,E2 -21293.68} C_VEL
LIN {X 0,Y 210.425,Z 286.887,A -85,B 0,C 180,E1 -21294.072,E2 -21294.072} C_VEL
LIN {X 0,Y 213.672,Z 299.218,A -85,B 0,C 180,E1 -21295.626,E2 -21295.626} C_VEL
LIN {X 0,Y 215.599,Z 309.948,A -85,B 0,C 180,E1 -21297.097,E2 -21297.097} C_VEL
LIN {X 0,Y 216.84,Z 320.812,A -85,B 0,C 180,E1 -21298.763,E2 -21298.763} C_VEL
LIN {X 0,Y 217.271,Z 330.579,A -85,B 0,C 180,E1 -21300.444,E2 -21300.444} C_VEL
LIN {X 0,Y 216.953,Z 341.256,A -85,B 0,C 180,E1 -21302.541,E2 -21302.541} C_VEL
LIN {X 0,Y 216.382,Z 347.768,A -85,B 0,C 180,E1 -21303.994,E2 -21303.994} C_VEL
LIN {X 0,Y 213.273,Z 357.978,A -85,B 0,C 180,E1 -21306.513,E2 -21306.513} C_VEL
LIN {X 0,Y 211.476,Z 361.898,A -85,B 0,C 180,E1 -21307.608,E2 -21307.608} C_VEL
LIN {X 0,Y 206.998,Z 367.845,A -85,B 0,C 180,E1 -21309.408,E2 -21309.408} C_VEL
LIN {X 0,Y 202.596,Z 373.119,A -85,B 0,C 180,E1 -21311.415,E2 -21311.415} C_VEL
LIN {X 0,Y 200.958,Z 375.985,A -85,B 0,C 180,E1 -21312.811,E2 -21312.811} C_VEL
LIN {X 0,Y 199.302,Z 380.949,A -85,B 0,C 180,E1 -21315.71,E2 -21315.71} C_VEL
LIN {X 0,Y 198.284,Z 384.969,A -85,B 0,C 180,E1 -21318.759,E2 -21318.759} C_VEL
LIN {X 0,Y 197.694,Z 387.948,A -85,B 0,C 180,E1 -21321.825,E2 -21321.825} C_VEL
LIN {X 0,Y 197.506,Z 390.059,A -85,B 0,C 180,E1 -21325.102,E2 -21325.102} C_VEL
LIN {X 0,Y 197.569,Z 391.022,A -85,B 0,C 180,E1 -21327.962,E2 -21327.962} C_VEL
LIN {X 0,Y 197.671,Z 391.246,A -85,B 0,C 180,E1 -21330,E2 -21330} C_VEL
LIN {X 0,Y 197.568,Z 391.012,A -85,B 0,C 180,E1 -21332.039,E2 -21332.039} C_VEL
LIN {X 0,Y 197.498,Z 390.053,A -85,B 0,C 180,E1 -21334.873,E2 -21334.873} C_VEL
LIN {X 0,Y 197.689,Z 387.917,A -85,B 0,C 180,E1 -21338.176,E2 -21338.176} C_VEL
LIN {X 0,Y 198.282,Z 384.923,A -85,B 0,C 180,E1 -21341.242,E2 -21341.242} C_VEL
LIN {X 0,Y 199.302,Z 380.886,A -85,B 0,C 180,E1 -21344.291,E2 -21344.291} C_VEL
LIN {X 0,Y 201.326,Z 374.711,A -85,B 0,C 180,E1 -21347.786,E2 -21347.786} C_VEL
LIN {X 0,Y 203.579,Z 367.834,A -85,B 0,C 180,E1 -21350.785,E2 -21350.785} C_VEL
LIN {X 0,Y 206.049,Z 359.625,A -85,B 0,C 180,E1 -21353.627,E2 -21353.627} C_VEL
LIN {X 0,Y 208.787,Z 351.088,A -85,B 0,C 180,E1 -21355.951,E2 -21355.951} C_VEL
LIN {X 0,Y 209.904,Z 346.08,A -85,B 0,C 180,E1 -21357.142,E2 -21357.142} C_VEL
LIN {X 0,Y 210.628,Z 336.109,A -85,B 0,C 180,E1 -21359.344,E2 -21359.344} C_VEL
LIN {X 0,Y 210.576,Z 325.193,A -85,B 0,C 180,E1 -21361.433,E2 -21361.433} C_VEL
LIN {X 0,Y 209.654,Z 313.72,A -85,B 0,C 180,E1 -21363.358,E2 -21363.358} C_VEL
LIN {X 0,Y 207.844,Z 302.156,A -85,B 0,C 180,E1 -21365.089,E2 -21365.089} C_VEL
LIN {X 0,Y 204.74,Z 289.548,A -85,B 0,C 180,E1 -21366.822,E2 -21366.822} C_VEL
LIN {X 0,Y 202.822,Z 283.361,A -85,B 0,C 180,E1 -21367.621,E2 -21367.621} C_VEL
LIN {X 0,Y 202.756,Z 282.878,A -85,B 0,C 180,E1 -21367.71,E2 -21367.71} C_VEL
LIN {X 0,Y 202.621,Z 279.672,A -85,B 0,C 180,E1 -21371.226,E2 -21371.226} C_VEL
LIN {X 0,Y 201.854,Z 275.749,A -85,B 0,C 180,E1 -21375.865,E2 -21375.865} C_VEL
LIN {X 0,Y 201.061,Z 271.698,A -85,B 0,C 180,E1 -21381.01,E2 -21381.01} C_VEL
LIN {X 0,Y 200.473,Z 268.207,A -85,B 0,C 180,E1 -21385.881,E2 -21385.881} C_VEL
LIN {X 0,Y 199.941,Z 265.221,A -85,B 0,C 180,E1 -21390.521,E2 -21390.521} C_VEL
LIN {X 0,Y 199.648,Z 263.618,A -85,B 0,C 180,E1 -21393.332,E2 -21393.332} C_VEL
LIN {X 0,Y 199.699,Z 263.614,A -85,B 0,C 180,E1 -21397.224,E2 -21397.224} C_VEL
LIN {X 0,Y 199.799,Z 263.598,A -85,B 0,C 180,E1 -21401.759,E2 -21401.759} C_VEL
LIN {X 0,Y 199.839,Z 263.592,A -85,B 0,C 180,E1 -21405.749,E2 -21405.749} C_VEL
LIN {X 0,Y 200.026,Z 263.569,A -85,B 0,C 180,E1 -21409.882,E2 -21409.882} C_VEL
LIN {X 0,Y 200.023,Z 263.571,A -85,B 0,C 180,E1 -21413.949,E2 -21413.949} C_VEL
LIN {X 0,Y 200.324,Z 263.531,A -85,B 0,C 180,E1 -21417.99,E2 -21417.99} C_VEL
LIN {X 0,Y 200.451,Z 263.514,A -85,B 0,C 180,E1 -21420,E2 -21420} C_VEL
LIN {X 0,Y 200.006,Z 263.571,A -85,B 0,C 180,E1 -21424.03,E2 -21424.03} C_VEL
LIN {X 0,Y 200.088,Z 263.56,A -85,B 0,C 180,E1 -21428.077,E2 -21428.077} C_VEL
LIN {X 0,Y 199.869,Z 263.585,A -85,B 0,C 180,E1 -21432.18,E2 -21432.18} C_VEL
LIN {X 0,Y 199.77,Z 263.601,A -85,B 0,C 180,E1 -21436.347,E2 -21436.347} C_VEL
LIN {X 0,Y 199.676,Z 263.611,A -85,B 0,C 180,E1 -21440.608,E2 -21440.608} C_VEL
LIN {X 0,Y 199.654,Z 263.616,A -85,B 0,C 180,E1 -21444.987,E2 -21444.987} C_VEL
LIN {X 0,Y 199.611,Z 263.62,A -85,B 0,C 180,E1 -21449.533,E2 -21449.533} C_VEL
LIN {X 0,Y 199.668,Z 263.615,A -85,B 0,C 180,E1 -21452.353,E2 -21452.353} C_VEL
LIN {X 0,Y 199.626,Z 263.615,A -85,B 0,C 180,E1 -21456.763,E2 -21456.763} C_VEL
LIN {X 0,Y 199.611,Z 263.616,A -85,B 0,C 180,E1 -21459.328,E2 -21459.328} C_VEL
LIN {X 0,Y 199.577,Z 263.622,A -85,B 0,C 180,E1 -21462.31,E2 -21462.31} C_VEL
LIN {X 0,Y 199.582,Z 263.622,A -85,B 0,C 180,E1 -21465.228,E2 -21465.228} C_VEL
LIN {X 0,Y 199.577,Z 263.626,A -85,B 0,C 180,E1 -21468.004,E2 -21468.004} C_VEL
LIN {X 0,Y 199.779,Z 264.833,A -85,B 0,C 180,E1 -21471.735,E2 -21471.735} C_VEL
LIN {X 0,Y 201.252,Z 268.376,A -85,B 0,C 180,E1 -21472.362,E2 -21472.362} C_VEL
LIN {X 0,Y 205.525,Z 276.951,A -85,B 0,C 180,E1 -21474.004,E2 -21474.004} C_VEL
LIN {X 0,Y 209.677,Z 287.847,A -85,B 0,C 180,E1 -21476.055,E2 -21476.055} C_VEL
LIN {X 0,Y 212.502,Z 298.152,A -85,B 0,C 180,E1 -21478.051,E2 -21478.051} C_VEL
LIN {X 0,Y 214.381,Z 308.236,A -85,B 0,C 180,E1 -21480.147,E2 -21480.147} C_VEL
LIN {X 0,Y 215.007,Z 314.08,A -85,B 0,C 180,E1 -21481.441,E2 -21481.441} C_VEL
LIN {X 0,Y 212.43,Z 324.322,A -85,B 0,C 180,E1 -21483.491,E2 -21483.491} C_VEL
LIN {X 0,Y 209.818,Z 333.369,A -85,B 0,C 180,E1 -21485.774,E2 -21485.774} C_VEL
LIN {X 0,Y 206.8,Z 342.24,A -85,B 0,C 180,E1 -21488.571,E2 -21488.571} C_VEL
LIN {X 0,Y 204.352,Z 349.366,A -85,B 0,C 180,E1 -21491.45,E2 -21491.45} C_VEL
LIN {X 0,Y 202.543,Z 354.171,A -85,B 0,C 180,E1 -21493.883,E2 -21493.883} C_VEL
LIN {X 0,Y 200.819,Z 358.834,A -85,B 0,C 180,E1 -21496.851,E2 -21496.851} C_VEL
LIN {X 0,Y 199.565,Z 362.394,A -85,B 0,C 180,E1 -21499.858,E2 -21499.858} C_VEL
LIN {X 0,Y 198.959,Z 364.231,A -85,B 0,C 180,E1 -21501.877,E2 -21501.877} C_VEL
LIN {X 0,Y 198.513,Z 365.609,A -85,B 0,C 180,E1 -21503.903,E2 -21503.903} C_VEL
LIN {X 0,Y 197.86,Z 367.2,A -85,B 0,C 180,E1 -21507.964,E2 -21507.964} C_VEL
LIN {X 0,Y 197.793,Z 367.427,A -85,B 0,C 180,E1 -21510,E2 -21510} C_VEL
LIN {X 0,Y 198.103,Z 366.648,A -85,B 0,C 180,E1 -21514.068,E2 -21514.068} C_VEL
LIN {X 0,Y 198.476,Z 365.684,A -85,B 0,C 180,E1 -21516.098,E2 -21516.098} C_VEL
LIN {X 0,Y 199.035,Z 363.923,A -85,B 0,C 180,E1 -21518.622,E2 -21518.622} C_VEL
LIN {X 0,Y 200.32,Z 360.304,A -85,B 0,C 180,E1 -21522.152,E2 -21522.152} C_VEL
LIN {X 0,Y 201.847,Z 356.077,A -85,B 0,C 180,E1 -21525.137,E2 -21525.137} C_VEL
LIN {X 0,Y 204.248,Z 349.665,A -85,B 0,C 180,E1 -21528.559,E2 -21528.559} C_VEL
LIN {X 0,Y 206.699,Z 342.614,A -85,B 0,C 180,E1 -21531.439,E2 -21531.439} C_VEL
LIN {X 0,Y 209.784,Z 333.812,A -85,B 0,C 180,E1 -21534.229,E2 -21534.229} C_VEL
LIN {X 0,Y 212.521,Z 324.266,A -85,B 0,C 180,E1 -21536.657,E2 -21536.657} C_VEL
LIN {X 0,Y 214.958,Z 314.782,A -85,B 0,C 180,E1 -21538.565,E2 -21538.565} C_VEL
LIN {X 0,Y 214.5,Z 308.77,A -85,B 0,C 180,E1 -21539.878,E2 -21539.878} C_VEL
LIN {X 0,Y 212.732,Z 299.079,A -85,B 0,C 180,E1 -21541.91,E2 -21541.91} C_VEL
LIN {X 0,Y 210.249,Z 289.722,A -85,B 0,C 180,E1 -21543.747,E2 -21543.747} C_VEL
LIN {X 0,Y 206.275,Z 278.634,A -85,B 0,C 180,E1 -21545.83,E2 -21545.83} C_VEL
LIN {X 0,Y 201.284,Z 268.359,A -85,B 0,C 180,E1 -21547.796,E2 -21547.796} C_VEL
LIN {X 0,Y 199.971,Z 265.652,A -85,B 0,C 180,E1 -21548.286,E2 -21548.286} C_VEL
LIN {X 0,Y 199.781,Z 264.85,A -85,B 0,C 180,E1 -21548.393,E2 -21548.393} C_VEL
LIN {X 0,Y 199.571,Z 263.626,A -85,B 0,C 180,E1 -21552.309,E2 -21552.309} C_VEL
LIN {X 0,Y 199.581,Z 263.625,A -85,B 0,C 180,E1 -21555.228,E2 -21555.228} C_VEL
LIN {X 0,Y 199.581,Z 263.624,A -85,B 0,C 180,E1 -21558.005,E2 -21558.005} C_VEL
LIN {X 0,Y 199.612,Z 263.62,A -85,B 0,C 180,E1 -21560.767,E2 -21560.767} C_VEL
LIN {X 0,Y 199.612,Z 263.619,A -85,B 0,C 180,E1 -21565.713,E2 -21565.713} C_VEL
LIN {X 0,Y 199.687,Z 263.609,A -85,B 0,C 180,E1 -21568.134,E2 -21568.134} C_VEL
LIN {X 0,Y 199.644,Z 263.616,A -85,B 0,C 180,E1 -21572.765,E2 -21572.765} C_VEL
LIN {X 0,Y 199.708,Z 263.607,A -85,B 0,C 180,E1 -21577.225,E2 -21577.225} C_VEL
LIN {X 0,Y 199.751,Z 263.599,A -85,B 0,C 180,E1 -21581.798,E2 -21581.798} C_VEL
LIN {X 0,Y 199.82,Z 263.591,A -85,B 0,C 180,E1 -21585.747,E2 -21585.747} C_VEL
LIN {X 0,Y 200.078,Z 263.56,A -85,B 0,C 180,E1 -21589.884,E2 -21589.884} C_VEL
LIN {X 0,Y 200.134,Z 263.554,A -85,B 0,C 180,E1 -21591.925,E2 -21591.925} C_VEL
LIN {X 0,Y 200.295,Z 263.535,A -85,B 0,C 180,E1 -21597.989,E2 -21597.989} C_VEL
LIN {X 0,Y 200.45,Z 263.512,A -85,B 0,C 180,E1 -21600,E2 -21600} C_VEL
LIN {X 0,Y 200.322,Z 263.533,A -85,B 0,C 180,E1 -21602.01,E2 -21602.01} C_VEL
LIN {X 0,Y 200.088,Z 263.562,A -85,B 0,C 180,E1 -21608.077,E2 -21608.077} C_VEL
LIN {X 0,Y 199.876,Z 263.585,A -85,B 0,C 180,E1 -21612.179,E2 -21612.179} C_VEL
LIN {X 0,Y 199.806,Z 263.597,A -85,B 0,C 180,E1 -21616.343,E2 -21616.343} C_VEL
LIN {X 0,Y 199.678,Z 263.614,A -85,B 0,C 180,E1 -21620.608,E2 -21620.608} C_VEL
LIN {X 0,Y 199.638,Z 263.622,A -85,B 0,C 180,E1 -21624.989,E2 -21624.989} C_VEL
LIN {X 0,Y 199.667,Z 263.648,A -85,B 0,C 180,E1 -21626.666,E2 -21626.666} C_VEL
LIN {X 0,Y 200.203,Z 266.731,A -85,B 0,C 180,E1 -21631.774,E2 -21631.774} C_VEL
LIN {X 0,Y 200.716,Z 269.968,A -85,B 0,C 180,E1 -21636.53,E2 -21636.53} C_VEL
LIN {X 0,Y 201.422,Z 273.721,A -85,B 0,C 180,E1 -21641.525,E2 -21641.525} C_VEL
LIN {X 0,Y 202.194,Z 277.325,A -85,B 0,C 180,E1 -21645.959,E2 -21645.959} C_VEL
LIN {X 0,Y 202.756,Z 280.58,A -85,B 0,C 180,E1 -21649.691,E2 -21649.691} C_VEL
LIN {X 0,Y 202.791,Z 283.178,A -85,B 0,C 180,E1 -21652.298,E2 -21652.298} C_VEL
LIN {X 0,Y 203.842,Z 286.592,A -85,B 0,C 180,E1 -21652.732,E2 -21652.732} C_VEL
LIN {X 0,Y 206.947,Z 297.949,A -85,B 0,C 180,E1 -21654.267,E2 -21654.267} C_VEL
LIN {X 0,Y 209.207,Z 310.073,A -85,B 0,C 180,E1 -21656.03,E2 -21656.03} C_VEL
LIN {X 0,Y 210.455,Z 322.163,A -85,B 0,C 180,E1 -21657.986,E2 -21657.986} C_VEL
LIN {X 0,Y 210.746,Z 333.026,A -85,B 0,C 180,E1 -21659.985,E2 -21659.985} C_VEL
LIN {X 0,Y 210.14,Z 344.097,A -85,B 0,C 180,E1 -21662.352,E2 -21662.352} C_VEL
LIN {X 0,Y 209.388,Z 349.304,A -85,B 0,C 180,E1 -21663.594,E2 -21663.594} C_VEL
LIN {X 0,Y 206.533,Z 358.21,A -85,B 0,C 180,E1 -21665.913,E2 -21665.913} C_VEL
LIN {X 0,Y 203.888,Z 366.752,A -85,B 0,C 180,E1 -21668.746,E2 -21668.746} C_VEL
LIN {X 0,Y 201.618,Z 373.776,A -85,B 0,C 180,E1 -21671.717,E2 -21671.717} C_VEL
LIN {X 0,Y 200.958,Z 375.985,A -85,B 0,C 180,E1 -21672.811,E2 -21672.811} C_VEL
LIN {X 0,Y 199.39,Z 378.669,A -85,B 0,C 180,E1 -21674.264,E2 -21674.264} C_VEL
LIN {X 0,Y 193.746,Z 383.733,A -85,B 0,C 180,E1 -21677.662,E2 -21677.662} C_VEL
LIN {X 0,Y 191.246,Z 386.027,A -85,B 0,C 180,E1 -21679.789,E2 -21679.789} C_VEL
LIN {X 0,Y 190.725,Z 386.981,A -85,B 0,C 180,E1 -21680.916,E2 -21680.916} C_VEL
LIN {X 0,Y 190.429,Z 389.738,A -85,B 0,C 180,E1 -21685.182,E2 -21685.182} C_VEL
LIN {X 0,Y 190.48,Z 390.595,A -85,B 0,C 180,E1 -21687.886,E2 -21687.886} C_VEL
LIN {X 0,Y 190.604,Z 390.82,A -85,B 0,C 180,E1 -21690,E2 -21690} C_VEL
LIN {X 0,Y 190.48,Z 390.585,A -85,B 0,C 180,E1 -21692.115,E2 -21692.115} C_VEL
LIN {X 0,Y 190.401,Z 389.762,A -85,B 0,C 180,E1 -21694.714,E2 -21694.714} C_VEL
LIN {X 0,Y 190.634,Z 387.487,A -85,B 0,C 180,E1 -21698.48,E2 -21698.48} C_VEL
LIN {X 0,Y 191.286,Z 384.492,A -85,B 0,C 180,E1 -21701.659,E2 -21701.659} C_VEL
LIN {X 0,Y 192.387,Z 380.455,A -85,B 0,C 180,E1 -21704.816,E2 -21704.816} C_VEL
LIN {X 0,Y 194.505,Z 374.277,A -85,B 0,C 180,E1 -21708.431,E2 -21708.431} C_VEL
LIN {X 0,Y 196.784,Z 367.738,A -85,B 0,C 180,E1 -21711.388,E2 -21711.388} C_VEL
LIN {X 0,Y 199.53,Z 359.192,A -85,B 0,C 180,E1 -21714.449,E2 -21714.449} C_VEL
LIN {X 0,Y 202.411,Z 350.656,A -85,B 0,C 180,E1 -21716.833,E2 -21716.833} C_VEL
LIN {X 0,Y 203.352,Z 345.631,A -85,B 0,C 180,E1 -21718.093,E2 -21718.093} C_VEL
LIN {X 0,Y 204.106,Z 335.652,A -85,B 0,C 180,E1 -21720.378,E2 -21720.378} C_VEL
LIN {X 0,Y 204.129,Z 325.271,A -85,B 0,C 180,E1 -21722.447,E2 -21722.447} C_VEL
LIN {X 0,Y 203.194,Z 313.15,A -85,B 0,C 180,E1 -21724.579,E2 -21724.579} C_VEL
LIN {X 0,Y 201.186,Z 300.698,A -85,B 0,C 180,E1 -21726.538,E2 -21726.538} C_VEL
LIN {X 0,Y 198.361,Z 289.792,A -85,B 0,C 180,E1 -21728.159,E2 -21728.159} C_VEL
LIN {X 0,Y 197.032,Z 286.128,A -85,B 0,C 180,E1 -21728.719,E2 -21728.719} C_VEL
LIN {X 0,Y 195.851,Z 283.008,A -85,B 0,C 180,E1 -21729.199,E2 -21729.199} C_VEL
LIN {X 0,Y 195.778,Z 282.383,A -85,B 0,C 180,E1 -21729.298,E2 -21729.298} C_VEL
LIN {X 0,Y 195.324,Z 279.147,A -85,B 0,C 180,E1 -21733.13,E2 -21733.13} C_VEL
LIN {X 0,Y 194.491,Z 275.258,A -85,B 0,C 180,E1 -21738.048,E2 -21738.048} C_VEL
LIN {X 0,Y 193.839,Z 271.7,A -85,B 0,C 180,E1 -21742.907,E2 -21742.907} C_VEL
LIN {X 0,Y 193.377,Z 268.975,A -85,B 0,C 180,E1 -21746.965,E2 -21746.965} C_VEL
LIN {X 0,Y 192.931,Z 266.074,A -85,B 0,C 180,E1 -21751.734,E2 -21751.734} C_VEL
LIN {X 0,Y 192.594,Z 264.498,A -85,B 0,C 180,E1 -21755.029,E2 -21755.029} C_VEL
LIN {X 0,Y 192.609,Z 264.496,A -85,B 0,C 180,E1 -21758.6,E2 -21758.6} C_VEL
LIN {X 0,Y 192.76,Z 264.476,A -85,B 0,C 180,E1 -21763.042,E2 -21763.042} C_VEL
LIN {X 0,Y 192.806,Z 264.469,A -85,B 0,C 180,E1 -21767.367,E2 -21767.367} C_VEL
LIN {X 0,Y 193.037,Z 264.442,A -85,B 0,C 180,E1 -21771.626,E2 -21771.626} C_VEL
LIN {X 0,Y 193.266,Z 264.41,A -85,B 0,C 180,E1 -21777.916,E2 -21777.916} C_VEL
LIN {X 0,Y 193.418,Z 264.391,A -85,B 0,C 180,E1 -21780,E2 -21780} C_VEL
LIN {X 0,Y 192.953,Z 264.45,A -85,B 0,C 180,E1 -21784.178,E2 -21784.178} C_VEL
LIN {X 0,Y 193.037,Z 264.439,A -85,B 0,C 180,E1 -21788.374,E2 -21788.374} C_VEL
LIN {X 0,Y 192.795,Z 264.468,A -85,B 0,C 180,E1 -21792.634,E2 -21792.634} C_VEL
LIN {X 0,Y 192.723,Z 264.478,A -85,B 0,C 180,E1 -21796.962,E2 -21796.962} C_VEL
LIN {X 0,Y 192.611,Z 264.493,A -85,B 0,C 180,E1 -21801.4,E2 -21801.4} C_VEL
LIN {X 0,Y 192.642,Z 264.487,A -85,B 0,C 180,E1 -21804.208,E2 -21804.208} C_VEL
LIN {X 0,Y 192.605,Z 264.493,A -85,B 0,C 180,E1 -21808.866,E2 -21808.866} C_VEL
LIN {X 0,Y 192.597,Z 264.493,A -85,B 0,C 180,E1 -21813.186,E2 -21813.186} C_VEL
LIN {X 0,Y 192.554,Z 264.499,A -85,B 0,C 180,E1 -21818.351,E2 -21818.351} C_VEL
LIN {X 0,Y 192.494,Z 264.506,A -85,B 0,C 180,E1 -21823.096,E2 -21823.096} C_VEL
LIN {X 0,Y 192.491,Z 264.506,A -85,B 0,C 180,E1 -21826.905,E2 -21826.905} C_VEL
LIN {X 0,Y 192.639,Z 265.329,A -85,B 0,C 180,E1 -21830.009,E2 -21830.009} C_VEL
LIN {X 0,Y 193.87,Z 268.36,A -85,B 0,C 180,E1 -21830.615,E2 -21830.615} C_VEL
LIN {X 0,Y 195.292,Z 270.538,A -85,B 0,C 180,E1 -21831.125,E2 -21831.125} C_VEL
LIN {X 0,Y 200.008,Z 280.339,A -85,B 0,C 180,E1 -21833.158,E2 -21833.158} C_VEL
LIN {X 0,Y 203.612,Z 290.236,A -85,B 0,C 180,E1 -21835.161,E2 -21835.161} C_VEL
LIN {X 0,Y 206.09,Z 299.44,A -85,B 0,C 180,E1 -21837.07,E2 -21837.07} C_VEL
LIN {X 0,Y 207.939,Z 309.686,A -85,B 0,C 180,E1 -21839.324,E2 -21839.324} C_VEL
LIN {X 0,Y 208.518,Z 315.783,A -85,B 0,C 180,E1 -21840.743,E2 -21840.743} C_VEL
LIN {X 0,Y 206.005,Z 325.14,A -85,B 0,C 180,E1 -21842.705,E2 -21842.705} C_VEL
LIN {X 0,Y 203.372,Z 333.799,A -85,B 0,C 180,E1 -21844.955,E2 -21844.955} C_VEL
LIN {X 0,Y 200.206,Z 342.67,A -85,B 0,C 180,E1 -21847.829,E2 -21847.829} C_VEL
LIN {X 0,Y 197.647,Z 349.794,A -85,B 0,C 180,E1 -21850.797,E2 -21850.797} C_VEL
LIN {X 0,Y 195.756,Z 354.599,A -85,B 0,C 180,E1 -21853.308,E2 -21853.308} C_VEL
LIN {X 0,Y 193.926,Z 359.262,A -85,B 0,C 180,E1 -21856.375,E2 -21856.375} C_VEL
LIN {X 0,Y 192.597,Z 362.822,A -85,B 0,C 180,E1 -21859.487,E2 -21859.487} C_VEL
LIN {X 0,Y 191.956,Z 364.658,A -85,B 0,C 180,E1 -21861.578,E2 -21861.578} C_VEL
LIN {X 0,Y 191.466,Z 366.036,A -85,B 0,C 180,E1 -21863.677,E2 -21863.677} C_VEL
LIN {X 0,Y 190.798,Z 367.626,A -85,B 0,C 180,E1 -21867.889,E2 -21867.889} C_VEL
LIN {X 0,Y 190.724,Z 367.853,A -85,B 0,C 180,E1 -21870,E2 -21870} C_VEL
LIN {X 0,Y 191.056,Z 367.073,A -85,B 0,C 180,E1 -21874.219,E2 -21874.219} C_VEL
LIN {X 0,Y 191.43,Z 366.111,A -85,B 0,C 180,E1 -21876.323,E2 -21876.323} C_VEL
LIN {X 0,Y 191.945,Z 364.584,A -85,B 0,C 180,E1 -21878.66,E2 -21878.66} C_VEL
LIN {X 0,Y 193.393,Z 360.73,A -85,B 0,C 180,E1 -21882.594,E2 -21882.594} C_VEL
LIN {X 0,Y 195.028,Z 356.502,A -85,B 0,C 180,E1 -21885.68,E2 -21885.68} C_VEL
LIN {X 0,Y 197.547,Z 350.09,A -85,B 0,C 180,E1 -21889.213,E2 -21889.213} C_VEL
LIN {X 0,Y 200.129,Z 343.038,A -85,B 0,C 180,E1 -21892.179,E2 -21892.179} C_VEL
LIN {X 0,Y 203.344,Z 334.236,A -85,B 0,C 180,E1 -21895.048,E2 -21895.048} C_VEL
LIN {X 0,Y 206.172,Z 324.845,A -85,B 0,C 180,E1 -21897.503,E2 -21897.503} C_VEL
LIN {X 0,Y 208.604,Z 315.215,A -85,B 0,C 180,E1 -21899.52,E2 -21899.52} C_VEL
LIN {X 0,Y 207.414,Z 305.658,A -85,B 0,C 180,E1 -21901.724,E2 -21901.724} C_VEL
LIN {X 0,Y 205.09,Z 295.152,A -85,B 0,C 180,E1 -21903.976,E2 -21903.976} C_VEL
LIN {X 0,Y 201.876,Z 285.045,A -85,B 0,C 180,E1 -21906.047,E2 -21906.047} C_VEL
LIN {X 0,Y 197.829,Z 275.746,A -85,B 0,C 180,E1 -21907.979,E2 -21907.979} C_VEL
LIN {X 0,Y 194.519,Z 269.274,A -85,B 0,C 180,E1 -21909.327,E2 -21909.327} C_VEL
LIN {X 0,Y 192.959,Z 266.643,A -85,B 0,C 180,E1 -21909.914,E2 -21909.914} C_VEL
LIN {X 0,Y 192.629,Z 265.352,A -85,B 0,C 180,E1 -21910.152,E2 -21910.152} C_VEL
LIN {X 0,Y 192.49,Z 264.506,A -85,B 0,C 180,E1 -21913.095,E2 -21913.095} C_VEL
LIN {X 0,Y 192.492,Z 264.502,A -85,B 0,C 180,E1 -21916.904,E2 -21916.904} C_VEL
LIN {X 0,Y 192.553,Z 264.499,A -85,B 0,C 180,E1 -21921.648,E2 -21921.648} C_VEL
LIN {X 0,Y 192.596,Z 264.494,A -85,B 0,C 180,E1 -21926.813,E2 -21926.813} C_VEL
LIN {X 0,Y 192.622,Z 264.489,A -85,B 0,C 180,E1 -21931.685,E2 -21931.685} C_VEL
LIN {X 0,Y 192.679,Z 264.484,A -85,B 0,C 180,E1 -21936.345,E2 -21936.345} C_VEL
LIN {X 0,Y 192.7,Z 264.477,A -85,B 0,C 180,E1 -21941.487,E2 -21941.487} C_VEL
LIN {X 0,Y 192.745,Z 264.472,A -85,B 0,C 180,E1 -21945.212,E2 -21945.212} C_VEL
LIN {X 0,Y 193.022,Z 264.438,A -85,B 0,C 180,E1 -21949.511,E2 -21949.511} C_VEL
LIN {X 0,Y 193.081,Z 264.433,A -85,B 0,C 180,E1 -21951.628,E2 -21951.628} C_VEL
LIN {X 0,Y 193.24,Z 264.414,A -85,B 0,C 180,E1 -21957.916,E2 -21957.916} C_VEL
LIN {X 0,Y 193.417,Z 264.388,A -85,B 0,C 180,E1 -21960,E2 -21960} C_VEL
LIN {X 0,Y 192.974,Z 264.446,A -85,B 0,C 180,E1 -21964.177,E2 -21964.177} C_VEL
LIN {X 0,Y 193.036,Z 264.44,A -85,B 0,C 180,E1 -21968.374,E2 -21968.374} C_VEL
LIN {X 0,Y 192.804,Z 264.465,A -85,B 0,C 180,E1 -21972.633,E2 -21972.633} C_VEL
LIN {X 0,Y 192.759,Z 264.474,A -85,B 0,C 180,E1 -21976.959,E2 -21976.959} C_VEL
LIN {X 0,Y 192.608,Z 264.493,A -85,B 0,C 180,E1 -21981.401,E2 -21981.401} C_VEL
LIN {X 0,Y 192.634,Z 264.623,A -85,B 0,C 180,E1 -21985.464,E2 -21985.464} C_VEL
LIN {X 0,Y 192.984,Z 266.619,A -85,B 0,C 180,E1 -21989.07,E2 -21989.07} C_VEL
LIN {X 0,Y 193.409,Z 269.226,A -85,B 0,C 180,E1 -21993.305,E2 -21993.305} C_VEL
LIN {X 0,Y 193.918,Z 272.443,A -85,B 0,C 180,E1 -21998.033,E2 -21998.033} C_VEL
LIN {X 0,Y 194.748,Z 276.342,A -85,B 0,C 180,E1 -22003.288,E2 -22003.288} C_VEL
LIN {X 0,Y 195.32,Z 279.211,A -85,B 0,C 180,E1 -22006.87,E2 -22006.87} C_VEL
LIN {X 0,Y 195.749,Z 282.454,A -85,B 0,C 180,E1 -22010.676,E2 -22010.676} C_VEL
LIN {X 0,Y 196.779,Z 285.725,A -85,B 0,C 180,E1 -22011.126,E2 -22011.126} C_VEL
LIN {X 0,Y 197.868,Z 288.382,A -85,B 0,C 180,E1 -22011.561,E2 -22011.561} C_VEL
LIN {X 0,Y 200.367,Z 296.999,A -85,B 0,C 180,E1 -22012.853,E2 -22012.853} C_VEL
LIN {X 0,Y 202.789,Z 309.694,A -85,B 0,C 180,E1 -22014.81,E2 -22014.81} C_VEL
LIN {X 0,Y 203.919,Z 320.71,A -85,B 0,C 180,E1 -22016.667,E2 -22016.667} C_VEL
LIN {X 0,Y 204.293,Z 331.214,A -85,B 0,C 180,E1 -22018.662,E2 -22018.662} C_VEL
LIN {X 0,Y 203.873,Z 340.919,A -85,B 0,C 180,E1 -22020.744,E2 -22020.744} C_VEL
LIN {X 0,Y 202.963,Z 348.874,A -85,B 0,C 180,E1 -22022.69,E2 -22022.69} C_VEL
LIN {X 0,Y 200.054,Z 357.741,A -85,B 0,C 180,E1 -22025.067,E2 -22025.067} C_VEL
LIN {X 0,Y 197.303,Z 365.948,A -85,B 0,C 180,E1 -22027.84,E2 -22027.84} C_VEL
LIN {X 0,Y 195.222,Z 372.317,A -85,B 0,C 180,E1 -22030.549,E2 -22030.549} C_VEL
LIN {X 0,Y 193.542,Z 377.209,A -85,B 0,C 180,E1 -22033.112,E2 -22033.112} C_VEL
LIN {X 0,Y 191.972,Z 381.972,A -85,B 0,C 180,E1 -22036.234,E2 -22036.234} C_VEL
LIN {X 0,Y 191.037,Z 385.629,A -85,B 0,C 180,E1 -22039.401,E2 -22039.401} C_VEL
LIN {X 0,Y 190.725,Z 386.981,A -85,B 0,C 180,E1 -22040.916,E2 -22040.916} C_VEL
LIN {X 0,Y 189.898,Z 388.336,A -85,B 0,C 180,E1 -22042.628,E2 -22042.628} C_VEL
LIN {X 0,Y 188.315,Z 389.343,A -85,B 0,C 180,E1 -22044.335,E2 -22044.335} C_VEL
LIN {X 0,Y 184.727,Z 390.366,A -85,B 0,C 180,E1 -22047.832,E2 -22047.832} C_VEL
LIN {X 0,Y 183.504,Z 390.364,A -85,B 0,C 180,E1 -22050.285,E2 -22050.285} C_VEL
LIN {X 0,Y 183.395,Z 390.158,A -85,B 0,C 180,E1 -22052.197,E2 -22052.197} C_VEL
LIN {X 0,Y 183.33,Z 389.43,A -85,B 0,C 180,E1 -22054.645,E2 -22054.645} C_VEL
LIN {X 0,Y 183.582,Z 387.057,A -85,B 0,C 180,E1 -22058.809,E2 -22058.809} C_VEL
LIN {X 0,Y 184.311,Z 384.062,A -85,B 0,C 180,E1 -22062.106,E2 -22062.106} C_VEL
LIN {X 0,Y 185.493,Z 380.023,A -85,B 0,C 180,E1 -22065.38,E2 -22065.38} C_VEL
LIN {X 0,Y 187.711,Z 373.844,A -85,B 0,C 180,E1 -22069.124,E2 -22069.124} C_VEL
LIN {X 0,Y 189.792,Z 368.358,A -85,B 0,C 180,E1 -22071.735,E2 -22071.735} C_VEL
LIN {X 0,Y 192.513,Z 360.259,A -85,B 0,C 180,E1 -22074.824,E2 -22074.824} C_VEL
LIN {X 0,Y 195.44,Z 352.034,A -85,B 0,C 180,E1 -22077.29,E2 -22077.29} C_VEL
LIN {X 0,Y 196.482,Z 348.247,A -85,B 0,C 180,E1 -22078.291,E2 -22078.291} C_VEL
LIN {X 0,Y 197.496,Z 339.21,A -85,B 0,C 180,E1 -22080.554,E2 -22080.554} C_VEL
LIN {X 0,Y 197.802,Z 328.203,A -85,B 0,C 180,E1 -22082.962,E2 -22082.962} C_VEL
LIN {X 0,Y 197.199,Z 316.507,A -85,B 0,C 180,E1 -22085.2,E2 -22085.2} C_VEL
LIN {X 0,Y 195.644,Z 304.684,A -85,B 0,C 180,E1 -22087.215,E2 -22087.215} C_VEL
LIN {X 0,Y 192.979,Z 293.166,A -85,B 0,C 180,E1 -22089.081,E2 -22089.081} C_VEL
LIN {X 0,Y 191.368,Z 288.751,A -85,B 0,C 180,E1 -22089.862,E2 -22089.862} C_VEL
LIN {X 0,Y 190.289,Z 286.197,A -85,B 0,C 180,E1 -22090.32,E2 -22090.32} C_VEL
LIN {X 0,Y 188.825,Z 282.954,A -85,B 0,C 180,E1 -22090.929,E2 -22090.929} C_VEL
LIN {X 0,Y 188.604,Z 281.882,A -85,B 0,C 180,E1 -22091.077,E2 -22091.077} C_VEL
LIN {X 0,Y 187.911,Z 278.562,A -85,B 0,C 180,E1 -22095.286,E2 -22095.286} C_VEL
LIN {X 0,Y 187.43,Z 276.117,A -85,B 0,C 180,E1 -22098.585,E2 -22098.585} C_VEL
LIN {X 0,Y 186.88,Z 273.007,A -85,B 0,C 180,E1 -22103.007,E2 -22103.007} C_VEL
LIN {X 0,Y 186.275,Z 269.757,A -85,B 0,C 180,E1 -22108.115,E2 -22108.115} C_VEL
LIN {X 0,Y 185.866,Z 266.97,A -85,B 0,C 180,E1 -22113.016,E2 -22113.016} C_VEL
LIN {X 0,Y 185.61,Z 265.368,A -85,B 0,C 180,E1 -22116.573,E2 -22116.573} C_VEL
LIN {X 0,Y 185.692,Z 265.356,A -85,B 0,C 180,E1 -22122.375,E2 -22122.375} C_VEL
LIN {X 0,Y 185.733,Z 265.35,A -85,B 0,C 180,E1 -22126.877,E2 -22126.877} C_VEL
LIN {X 0,Y 185.984,Z 265.319,A -85,B 0,C 180,E1 -22131.306,E2 -22131.306} C_VEL
LIN {X 0,Y 186.21,Z 265.289,A -85,B 0,C 180,E1 -22137.837,E2 -22137.837} C_VEL
LIN {X 0,Y 186.384,Z 265.267,A -85,B 0,C 180,E1 -22140,E2 -22140} C_VEL
LIN {X 0,Y 185.901,Z 265.328,A -85,B 0,C 180,E1 -22144.336,E2 -22144.336} C_VEL
LIN {X 0,Y 185.984,Z 265.316,A -85,B 0,C 180,E1 -22148.694,E2 -22148.694} C_VEL
LIN {X 0,Y 185.721,Z 265.351,A -85,B 0,C 180,E1 -22153.124,E2 -22153.124} C_VEL
LIN {X 0,Y 185.66,Z 265.355,A -85,B 0,C 180,E1 -22157.628,E2 -22157.628} C_VEL
LIN {X 0,Y 185.574,Z 265.37,A -85,B 0,C 180,E1 -22162.254,E2 -22162.254} C_VEL
LIN {X 0,Y 185.58,Z 265.369,A -85,B 0,C 180,E1 -22164.646,E2 -22164.646} C_VEL
LIN {X 0,Y 185.546,Z 265.373,A -85,B 0,C 180,E1 -22169.499,E2 -22169.499} C_VEL
LIN {X 0,Y 185.501,Z 265.377,A -85,B 0,C 180,E1 -22174.632,E2 -22174.632} C_VEL
LIN {X 0,Y 185.509,Z 265.377,A -85,B 0,C 180,E1 -22177.313,E2 -22177.313} C_VEL
LIN {X 0,Y 185.474,Z 265.382,A -85,B 0,C 180,E1 -22180.725,E2 -22180.725} C_VEL
LIN {X 0,Y 185.48,Z 265.382,A -85,B 0,C 180,E1 -22183.951,E2 -22183.951} C_VEL
LIN {X 0,Y 185.458,Z 265.398,A -85,B 0,C 180,E1 -22186.99,E2 -22186.99} C_VEL
LIN {X 0,Y 185.536,Z 266.04,A -85,B 0,C 180,E1 -22188.234,E2 -22188.234} C_VEL
LIN {X 0,Y 186.576,Z 268.663,A -85,B 0,C 180,E1 -22188.727,E2 -22188.727} C_VEL
LIN {X 0,Y 188.408,Z 271.382,A -85,B 0,C 180,E1 -22189.439,E2 -22189.439} C_VEL
LIN {X 0,Y 192.15,Z 278.552,A -85,B 0,C 180,E1 -22191.113,E2 -22191.113} C_VEL
LIN {X 0,Y 195.962,Z 287.541,A -85,B 0,C 180,E1 -22193.118,E2 -22193.118} C_VEL
LIN {X 0,Y 198.898,Z 297.248,A -85,B 0,C 180,E1 -22195.239,E2 -22195.239} C_VEL
LIN {X 0,Y 200.983,Z 307.132,A -85,B 0,C 180,E1 -22197.493,E2 -22197.493} C_VEL
LIN {X 0,Y 202.084,Z 316.234,A -85,B 0,C 180,E1 -22199.716,E2 -22199.716} C_VEL
LIN {X 0,Y 201.403,Z 319.721,A -85,B 0,C 180,E1 -22200.468,E2 -22200.468} C_VEL
LIN {X 0,Y 198.705,Z 328.986,A -85,B 0,C 180,E1 -22202.625,E2 -22202.625} C_VEL
LIN {X 0,Y 195.815,Z 337.431,A -85,B 0,C 180,E1 -22205.056,E2 -22205.056} C_VEL
LIN {X 0,Y 192.733,Z 345.637,A -85,B 0,C 180,E1 -22208.051,E2 -22208.051} C_VEL
LIN {X 0,Y 190.533,Z 351.245,A -85,B 0,C 180,E1 -22210.611,E2 -22210.611} C_VEL
LIN {X 0,Y 188.278,Z 356.708,A -85,B 0,C 180,E1 -22213.742,E2 -22213.742} C_VEL
LIN {X 0,Y 186.485,Z 360.991,A -85,B 0,C 180,E1 -22216.931,E2 -22216.931} C_VEL
LIN {X 0,Y 185.069,Z 364.781,A -85,B 0,C 180,E1 -22220.879,E2 -22220.879} C_VEL
LIN {X 0,Y 184.426,Z 366.463,A -85,B 0,C 180,E1 -22223.435,E2 -22223.435} C_VEL
LIN {X 0,Y 184.02,Z 367.446,A -85,B 0,C 180,E1 -22225.619,E2 -22225.619} C_VEL
LIN {X 0,Y 183.658,Z 368.278,A -85,B 0,C 180,E1 -22230,E2 -22230} C_VEL
LIN {X 0,Y 184.012,Z 367.498,A -85,B 0,C 180,E1 -22234.381,E2 -22234.381} C_VEL
LIN {X 0,Y 184.389,Z 366.537,A -85,B 0,C 180,E1 -22236.566,E2 -22236.566} C_VEL
LIN {X 0,Y 184.879,Z 365.193,A -85,B 0,C 180,E1 -22238.746,E2 -22238.746} C_VEL
LIN {X 0,Y 186.016,Z 362.345,A -85,B 0,C 180,E1 -22241.993,E2 -22241.993} C_VEL
LIN {X 0,Y 187.566,Z 358.48,A -85,B 0,C 180,E1 -22245.206,E2 -22245.206} C_VEL
LIN {X 0,Y 189.638,Z 353.485,A -85,B 0,C 180,E1 -22248.361,E2 -22248.361} C_VEL
LIN {X 0,Y 192.197,Z 347.186,A -85,B 0,C 180,E1 -22251.448,E2 -22251.448} C_VEL
LIN {X 0,Y 195.192,Z 339.302,A -85,B 0,C 180,E1 -22254.46,E2 -22254.46} C_VEL
LIN {X 0,Y 198.08,Z 331.254,A -85,B 0,C 180,E1 -22256.896,E2 -22256.896} C_VEL
LIN {X 0,Y 200.992,Z 321.447,A -85,B 0,C 180,E1 -22259.31,E2 -22259.31} C_VEL
LIN {X 0,Y 202.163,Z 316.858,A -85,B 0,C 180,E1 -22260.27,E2 -22260.27} C_VEL
LIN {X 0,Y 201.052,Z 307.064,A -85,B 0,C 180,E1 -22262.665,E2 -22262.665} C_VEL
LIN {X 0,Y 199.05,Z 297.644,A -85,B 0,C 180,E1 -22264.824,E2 -22264.824} C_VEL
LIN {X 0,Y 196.286,Z 288.412,A -85,B 0,C 180,E1 -22266.85,E2 -22266.85} C_VEL
LIN {X 0,Y 191.754,Z 277.642,A -85,B 0,C 180,E1 -22269.261,E2 -22269.261} C_VEL
LIN {X 0,Y 189.479,Z 273.489,A -85,B 0,C 180,E1 -22270.255,E2 -22270.255} C_VEL
LIN {X 0,Y 187.541,Z 269.962,A -85,B 0,C 180,E1 -22271.084,E2 -22271.084} C_VEL
LIN {X 0,Y 185.817,Z 267.151,A -85,B 0,C 180,E1 -22271.785,E2 -22271.785} C_VEL
LIN {X 0,Y 185.516,Z 265.909,A -85,B 0,C 180,E1 -22271.991,E2 -22271.991} C_VEL
LIN {X 0,Y 185.46,Z 265.38,A -85,B 0,C 180,E1 -22273.945,E2 -22273.945} C_VEL
LIN {X 0,Y 185.473,Z 265.381,A -85,B 0,C 180,E1 -22279.275,E2 -22279.275} C_VEL
LIN {X 0,Y 185.508,Z 265.378,A -85,B 0,C 180,E1 -22282.711,E2 -22282.711} C_VEL
LIN {X 0,Y 185.532,Z 265.372,A -85,B 0,C 180,E1 -22287.972,E2 -22287.972} C_VEL
LIN {X 0,Y 185.548,Z 265.372,A -85,B 0,C 180,E1 -22290.595,E2 -22290.595} C_VEL
LIN {X 0,Y 185.581,Z 265.366,A -85,B 0,C 180,E1 -22295.381,E2 -22295.381} C_VEL
LIN {X 0,Y 185.635,Z 265.358,A -85,B 0,C 180,E1 -22301.17,E2 -22301.17} C_VEL
LIN {X 0,Y 185.673,Z 265.354,A -85,B 0,C 180,E1 -22304.635,E2 -22304.635} C_VEL
LIN {X 0,Y 185.94,Z 265.32,A -85,B 0,C 180,E1 -22309.335,E2 -22309.335} C_VEL
LIN {X 0,Y 186.031,Z 265.312,A -85,B 0,C 180,E1 -22311.308,E2 -22311.308} C_VEL
LIN {X 0,Y 186.186,Z 265.293,A -85,B 0,C 180,E1 -22317.837,E2 -22317.837} C_VEL
LIN {X 0,Y 186.383,Z 265.264,A -85,B 0,C 180,E1 -22320,E2 -22320} C_VEL
LIN {X 0,Y 185.921,Z 265.325,A -85,B 0,C 180,E1 -22324.336,E2 -22324.336} C_VEL
LIN {X 0,Y 185.983,Z 265.317,A -85,B 0,C 180,E1 -22328.694,E2 -22328.694} C_VEL
LIN {X 0,Y 185.731,Z 265.347,A -85,B 0,C 180,E1 -22333.123,E2 -22333.123} C_VEL
LIN {X 0,Y 185.691,Z 265.352,A -85,B 0,C 180,E1 -22337.625,E2 -22337.625} C_VEL
LIN {X 0,Y 185.617,Z 265.366,A -85,B 0,C 180,E1 -22343.722,E2 -22343.722} C_VEL
LIN {X 0,Y 186.081,Z 268.359,A -85,B 0,C 180,E1 -22349.406,E2 -22349.406} C_VEL
LIN {X 0,Y 186.531,Z 271.4,A -85,B 0,C 180,E1 -22354.414,E2 -22354.414} C_VEL
LIN {X 0,Y 186.931,Z 273.667,A -85,B 0,C 180,E1 -22357.858,E2 -22357.858} C_VEL
LIN {X 0,Y 187.594,Z 276.902,A -85,B 0,C 180,E1 -22362.404,E2 -22362.404} C_VEL
LIN {X 0,Y 188.259,Z 280.028,A -85,B 0,C 180,E1 -22366.513,E2 -22366.513} C_VEL
LIN {X 0,Y 188.591,Z 281.902,A -85,B 0,C 180,E1 -22368.85,E2 -22368.85} C_VEL
LIN {X 0,Y 189.767,Z 285.292,A -85,B 0,C 180,E1 -22369.405,E2 -22369.405} C_VEL
LIN {X 0,Y 191.041,Z 287.902,A -85,B 0,C 180,E1 -22369.92,E2 -22369.92} C_VEL
LIN {X 0,Y 193.309,Z 294.052,A -85,B 0,C 180,E1 -22371.004,E2 -22371.004} C_VEL
LIN {X 0,Y 195.933,Z 306.322,A -85,B 0,C 180,E1 -22372.983,E2 -22372.983} C_VEL
LIN {X 0,Y 197.21,Z 316.224,A -85,B 0,C 180,E1 -22374.696,E2 -22374.696} C_VEL
LIN {X 0,Y 197.832,Z 327.176,A -85,B 0,C 180,E1 -22376.775,E2 -22376.775} C_VEL
LIN {X 0,Y 197.704,Z 336.47,A -85,B 0,C 180,E1 -22378.758,E2 -22378.758} C_VEL
LIN {X 0,Y 196.796,Z 346.45,A -85,B 0,C 180,E1 -22381.177,E2 -22381.177} C_VEL
LIN {X 0,Y 196.066,Z 350.403,A -85,B 0,C 180,E1 -22382.226,E2 -22382.226} C_VEL
LIN {X 0,Y 193.055,Z 358.902,A -85,B 0,C 180,E1 -22384.675,E2 -22384.675} C_VEL
LIN {X 0,Y 190.186,Z 367.134,A -85,B 0,C 180,E1 -22387.701,E2 -22387.701} C_VEL
LIN {X 0,Y 187.729,Z 373.939,A -85,B 0,C 180,E1 -22390.879,E2 -22390.879} C_VEL
LIN {X 0,Y 185.493,Z 380.091,A -85,B 0,C 180,E1 -22394.62,E2 -22394.62} C_VEL
LIN {X 0,Y 184.313,Z 384.111,A -85,B 0,C 180,E1 -22397.894,E2 -22397.894} C_VEL
LIN {X 0,Y 183.586,Z 387.09,A -85,B 0,C 180,E1 -22401.192,E2 -22401.192} C_VEL
LIN {X 0,Y 183.329,Z 389.447,A -85,B 0,C 180,E1 -22405.36,E2 -22405.36} C_VEL
LIN {X 0,Y 183.395,Z 390.168,A -85,B 0,C 180,E1 -22407.804,E2 -22407.804} C_VEL
LIN {X 0,Y 183.504,Z 390.364,A -85,B 0,C 180,E1 -22410.285,E2 -22410.285} C_VEL
LIN {X 0,Y 182.676,Z 390.135,A -85,B 0,C 180,E1 -22412.112,E2 -22412.112} C_VEL
LIN {X 0,Y 179.739,Z 389.08,A -85,B 0,C 180,E1 -22415.094,E2 -22415.094} C_VEL
LIN {X 0,Y 177.457,Z 387.754,A -85,B 0,C 180,E1 -22417.518,E2 -22417.518} C_VEL
LIN {X 0,Y 176.664,Z 386.46,A -85,B 0,C 180,E1 -22419.381,E2 -22419.381} C_VEL
LIN {X 0,Y 176.693,Z 385.928,A -85,B 0,C 180,E1 -22420.004,E2 -22420.004} C_VEL
LIN {X 0,Y 177.683,Z 382.38,A -85,B 0,C 180,E1 -22423.729,E2 -22423.729} C_VEL
LIN {X 0,Y 179.273,Z 377.982,A -85,B 0,C 180,E1 -22427.099,E2 -22427.099} C_VEL
LIN {X 0,Y 181.399,Z 372.393,A -85,B 0,C 180,E1 -22430.408,E2 -22430.408} C_VEL
LIN {X 0,Y 183.9,Z 365.801,A -85,B 0,C 180,E1 -22433.48,E2 -22433.48} C_VEL
LIN {X 0,Y 186.624,Z 358.328,A -85,B 0,C 180,E1 -22436.263,E2 -22436.263} C_VEL
LIN {X 0,Y 189.684,Z 349.783,A -85,B 0,C 180,E1 -22438.795,E2 -22438.795} C_VEL
LIN {X 0,Y 190.974,Z 339.933,A -85,B 0,C 180,E1 -22441.412,E2 -22441.412} C_VEL
LIN {X 0,Y 191.457,Z 329.254,A -85,B 0,C 180,E1 -22443.873,E2 -22443.873} C_VEL
LIN {X 0,Y 191.071,Z 318.601,A -85,B 0,C 180,E1 -22446.052,E2 -22446.052} C_VEL
LIN {X 0,Y 189.879,Z 307.725,A -85,B 0,C 180,E1 -22448.063,E2 -22448.063} C_VEL
LIN {X 0,Y 187.485,Z 296.188,A -85,B 0,C 180,E1 -22450.097,E2 -22450.097} C_VEL
LIN {X 0,Y 185.229,Z 290.152,A -85,B 0,C 180,E1 -22451.289,E2 -22451.289} C_VEL
LIN {X 0,Y 183.344,Z 286.049,A -85,B 0,C 180,E1 -22452.153,E2 -22452.153} C_VEL
LIN {X 0,Y 181.658,Z 282.896,A -85,B 0,C 180,E1 -22452.882,E2 -22452.882} C_VEL
LIN {X 0,Y 181.288,Z 281.289,A -85,B 0,C 180,E1 -22453.153,E2 -22453.153} C_VEL
LIN {X 0,Y 180.468,Z 277.391,A -85,B 0,C 180,E1 -22458.545,E2 -22458.545} C_VEL
LIN {X 0,Y 179.732,Z 273.691,A -85,B 0,C 180,E1 -22464.088,E2 -22464.088} C_VEL
LIN {X 0,Y 179.205,Z 270.535,A -85,B 0,C 180,E1 -22469.348,E2 -22469.348} C_VEL
LIN {X 0,Y 178.777,Z 267.865,A -85,B 0,C 180,E1 -22474.378,E2 -22474.378} C_VEL
LIN {X 0,Y 178.517,Z 266.25,A -85,B 0,C 180,E1 -22478.037,E2 -22478.037} C_VEL
LIN {X 0,Y 178.652,Z 266.232,A -85,B 0,C 180,E1 -22481.657,E2 -22481.657} C_VEL
LIN {X 0,Y 178.661,Z 266.23,A -85,B 0,C 180,E1 -22486.348,E2 -22486.348} C_VEL
LIN {X 0,Y 178.913,Z 266.199,A -85,B 0,C 180,E1 -22490.96,E2 -22490.96} C_VEL
LIN {X 0,Y 179.155,Z 266.168,A -85,B 0,C 180,E1 -22497.752,E2 -22497.752} C_VEL
LIN {X 0,Y 179.349,Z 266.143,A -85,B 0,C 180,E1 -22500,E2 -22500} C_VEL
LIN {X 0,Y 178.85,Z 266.207,A -85,B 0,C 180,E1 -22504.508,E2 -22504.508} C_VEL
LIN {X 0,Y 178.913,Z 266.197,A -85,B 0,C 180,E1 -22509.04,E2 -22509.04} C_VEL
LIN {X 0,Y 178.647,Z 266.232,A -85,B 0,C 180,E1 -22513.653,E2 -22513.653} C_VEL
LIN {X 0,Y 178.594,Z 266.24,A -85,B 0,C 180,E1 -22519.186,E2 -22519.186} C_VEL
LIN {X 0,Y 178.518,Z 266.248,A -85,B 0,C 180,E1 -22525.111,E2 -22525.111} C_VEL
LIN {X 0,Y 178.463,Z 266.254,A -85,B 0,C 180,E1 -22530.794,E2 -22530.794} C_VEL
LIN {X 0,Y 178.486,Z 266.254,A -85,B 0,C 180,E1 -22534.218,E2 -22534.218} C_VEL
LIN {X 0,Y 178.399,Z 266.258,A -85,B 0,C 180,E1 -22539.074,E2 -22539.074} C_VEL
LIN {X 0,Y 178.401,Z 266.26,A -85,B 0,C 180,E1 -22542.045,E2 -22542.045} C_VEL
LIN {X 0,Y 178.445,Z 266.491,A -85,B 0,C 180,E1 -22546.157,E2 -22546.157} C_VEL
LIN {X 0,Y 179.515,Z 269.284,A -85,B 0,C 180,E1 -22546.72,E2 -22546.72} C_VEL
LIN {X 0,Y 181.258,Z 271.691,A -85,B 0,C 180,E1 -22547.451,E2 -22547.451} C_VEL
LIN {X 0,Y 186.176,Z 280.801,A -85,B 0,C 180,E1 -22549.824,E2 -22549.824} C_VEL
LIN {X 0,Y 190.279,Z 290.753,A -85,B 0,C 180,E1 -22552.241,E2 -22552.241} C_VEL
LIN {X 0,Y 193.03,Z 300.326,A -85,B 0,C 180,E1 -22554.507,E2 -22554.507} C_VEL
LIN {X 0,Y 194.921,Z 310.45,A -85,B 0,C 180,E1 -22556.989,E2 -22556.989} C_VEL
LIN {X 0,Y 195.671,Z 317.841,A -85,B 0,C 180,E1 -22558.914,E2 -22558.914} C_VEL
LIN {X 0,Y 195.27,Z 320.152,A -85,B 0,C 180,E1 -22559.444,E2 -22559.444} C_VEL
LIN {X 0,Y 192.45,Z 329.416,A -85,B 0,C 180,E1 -22561.657,E2 -22561.657} C_VEL
LIN {X 0,Y 189.425,Z 337.86,A -85,B 0,C 180,E1 -22564.154,E2 -22564.154} C_VEL
LIN {X 0,Y 186.186,Z 346.066,A -85,B 0,C 180,E1 -22567.237,E2 -22567.237} C_VEL
LIN {X 0,Y 183.856,Z 351.674,A -85,B 0,C 180,E1 -22569.877,E2 -22569.877} C_VEL
LIN {X 0,Y 181.487,Z 357.136,A -85,B 0,C 180,E1 -22573.116,E2 -22573.116} C_VEL
LIN {X 0,Y 179.579,Z 361.42,A -85,B 0,C 180,E1 -22576.419,E2 -22576.419} C_VEL
LIN {X 0,Y 177.992,Z 365.426,A -85,B 0,C 180,E1 -22580.797,E2 -22580.797} C_VEL
LIN {X 0,Y 177.392,Z 366.89,A -85,B 0,C 180,E1 -22583.174,E2 -22583.174} C_VEL
LIN {X 0,Y 176.979,Z 367.871,A -85,B 0,C 180,E1 -22585.444,E2 -22585.444} C_VEL
LIN {X 0,Y 176.593,Z 368.704,A -85,B 0,C 180,E1 -22590,E2 -22590} C_VEL
LIN {X 0,Y 176.97,Z 367.923,A -85,B 0,C 180,E1 -22594.555,E2 -22594.555} C_VEL
LIN {X 0,Y 177.804,Z 365.792,A -85,B 0,C 180,E1 -22598.82,E2 -22598.82} C_VEL
LIN {X 0,Y 179.097,Z 362.77,A -85,B 0,C 180,E1 -22602.464,E2 -22602.464} C_VEL
LIN {X 0,Y 180.726,Z 358.906,A -85,B 0,C 180,E1 -22605.796,E2 -22605.796} C_VEL
LIN {X 0,Y 182.928,Z 353.91,A -85,B 0,C 180,E1 -22609.06,E2 -22609.06} C_VEL
LIN {X 0,Y 185.61,Z 347.611,A -85,B 0,C 180,E1 -22612.249,E2 -22612.249} C_VEL
LIN {X 0,Y 188.783,Z 339.725,A -85,B 0,C 180,E1 -22615.348,E2 -22615.348} C_VEL
LIN {X 0,Y 191.795,Z 331.677,A -85,B 0,C 180,E1 -22617.853,E2 -22617.853} C_VEL
LIN {X 0,Y 194.851,Z 321.869,A -85,B 0,C 180,E1 -22620.329,E2 -22620.329} C_VEL
LIN {X 0,Y 195.771,Z 318.444,A -85,B 0,C 180,E1 -22621.067,E2 -22621.067} C_VEL
LIN {X 0,Y 194.721,Z 308.578,A -85,B 0,C 180,E1 -22623.632,E2 -22623.632} C_VEL
LIN {X 0,Y 192.567,Z 298.27,A -85,B 0,C 180,E1 -22626.149,E2 -22626.149} C_VEL
LIN {X 0,Y 189.955,Z 289.771,A -85,B 0,C 180,E1 -22628.16,E2 -22628.16} C_VEL
LIN {X 0,Y 185.311,Z 278.942,A -85,B 0,C 180,E1 -22630.813,E2 -22630.813} C_VEL
LIN {X 0,Y 182.277,Z 273.74,A -85,B 0,C 180,E1 -22632.232,E2 -22632.232} C_VEL
LIN {X 0,Y 180.69,Z 270.778,A -85,B 0,C 180,E1 -22632.983,E2 -22632.983} C_VEL
LIN {X 0,Y 178.983,Z 268.31,A -85,B 0,C 180,E1 -22633.718,E2 -22633.718} C_VEL
LIN {X 0,Y 178.453,Z 266.467,A -85,B 0,C 180,E1 -22634.049,E2 -22634.049} C_VEL
LIN {X 0,Y 178.405,Z 266.263,A -85,B 0,C 180,E1 -22638.459,E2 -22638.459} C_VEL
LIN {X 0,Y 178.424,Z 266.259,A -85,B 0,C 180,E1 -22643.783,E2 -22643.783} C_VEL
LIN {X 0,Y 178.485,Z 266.251,A -85,B 0,C 180,E1 -22646.546,E2 -22646.546} C_VEL
LIN {X 0,Y 178.445,Z 266.254,A -85,B 0,C 180,E1 -22651.795,E2 -22651.795} C_VEL
LIN {X 0,Y 178.516,Z 266.244,A -85,B 0,C 180,E1 -22654.889,E2 -22654.889} C_VEL
LIN {X 0,Y 178.592,Z 266.237,A -85,B 0,C 180,E1 -22660.814,E2 -22660.814} C_VEL
LIN {X 0,Y 178.652,Z 266.229,A -85,B 0,C 180,E1 -22666.347,E2 -22666.347} C_VEL
LIN {X 0,Y 178.979,Z 266.192,A -85,B 0,C 180,E1 -22670.963,E2 -22670.963} C_VEL
LIN {X 0,Y 179.134,Z 266.171,A -85,B 0,C 180,E1 -22677.751,E2 -22677.751} C_VEL
LIN {X 0,Y 179.348,Z 266.141,A -85,B 0,C 180,E1 -22680,E2 -22680} C_VEL
LIN {X 0,Y 178.868,Z 266.205,A -85,B 0,C 180,E1 -22684.507,E2 -22684.507} C_VEL
LIN {X 0,Y 178.912,Z 266.197,A -85,B 0,C 180,E1 -22689.04,E2 -22689.04} C_VEL
LIN {X 0,Y 178.659,Z 266.23,A -85,B 0,C 180,E1 -22693.652,E2 -22693.652} C_VEL
LIN {X 0,Y 178.622,Z 266.235,A -85,B 0,C 180,E1 -22699.214,E2 -22699.214} C_VEL
LIN {X 0,Y 178.559,Z 266.479,A -85,B 0,C 180,E1 -22702.566,E2 -22702.566} C_VEL
LIN {X 0,Y 178.992,Z 269.206,A -85,B 0,C 180,E1 -22708.11,E2 -22708.11} C_VEL
LIN {X 0,Y 179.445,Z 272.132,A -85,B 0,C 180,E1 -22713.251,E2 -22713.251} C_VEL
LIN {X 0,Y 180.03,Z 275.559,A -85,B 0,C 180,E1 -22718.67,E2 -22718.67} C_VEL
LIN {X 0,Y 180.603,Z 278.063,A -85,B 0,C 180,E1 -22722.323,E2 -22722.323} C_VEL
LIN {X 0,Y 181.281,Z 281.339,A -85,B 0,C 180,E1 -22726.799,E2 -22726.799} C_VEL
LIN {X 0,Y 182.397,Z 284.608,A -85,B 0,C 180,E1 -22727.381,E2 -22727.381} C_VEL
LIN {X 0,Y 183.992,Z 287.295,A -85,B 0,C 180,E1 -22728.042,E2 -22728.042} C_VEL
LIN {X 0,Y 187.061,Z 294.565,A -85,B 0,C 180,E1 -22729.536,E2 -22729.536} C_VEL
LIN {X 0,Y 189.283,Z 304.196,A -85,B 0,C 180,E1 -22731.235,E2 -22731.235} C_VEL
LIN {X 0,Y 190.901,Z 315.583,A -85,B 0,C 180,E1 -22733.314,E2 -22733.314} C_VEL
LIN {X 0,Y 191.493,Z 327.284,A -85,B 0,C 180,E1 -22735.643,E2 -22735.643} C_VEL
LIN {X 0,Y 191.171,Z 338.411,A -85,B 0,C 180,E1 -22738.17,E2 -22738.17} C_VEL
LIN {X 0,Y 190.057,Z 347.998,A -85,B 0,C 180,E1 -22740.662,E2 -22740.662} C_VEL
LIN {X 0,Y 189.147,Z 351.779,A -85,B 0,C 180,E1 -22741.723,E2 -22741.723} C_VEL
LIN {X 0,Y 186.059,Z 359.973,A -85,B 0,C 180,E1 -22744.254,E2 -22744.254} C_VEL
LIN {X 0,Y 183.107,Z 368.041,A -85,B 0,C 180,E1 -22747.43,E2 -22747.43} C_VEL
LIN {X 0,Y 180.647,Z 374.516,A -85,B 0,C 180,E1 -22750.69,E2 -22750.69} C_VEL
LIN {X 0,Y 178.627,Z 379.663,A -85,B 0,C 180,E1 -22754.014,E2 -22754.014} C_VEL
LIN {X 0,Y 177.332,Z 383.682,A -85,B 0,C 180,E1 -22757.41,E2 -22757.41} C_VEL
LIN {X 0,Y 176.556,Z 386.663,A -85,B 0,C 180,E1 -22760.838,E2 -22760.838} C_VEL
LIN {X 0,Y 176.306,Z 388.088,A -85,B 0,C 180,E1 -22763.132,E2 -22763.132} C_VEL
LIN {X 0,Y 176.262,Z 389.113,A -85,B 0,C 180,E1 -22765.426,E2 -22765.426} C_VEL
LIN {X 0,Y 176.313,Z 389.742,A -85,B 0,C 180,E1 -22767.716,E2 -22767.716} C_VEL
LIN {X 0,Y 176.448,Z 389.949,A -85,B 0,C 180,E1 -22770.193,E2 -22770.193} C_VEL
LIN {X 0,Y 176.311,Z 389.731,A -85,B 0,C 180,E1 -22772.285,E2 -22772.285} C_VEL
LIN {X 0,Y 176.262,Z 389.096,A -85,B 0,C 180,E1 -22774.574,E2 -22774.574} C_VEL
LIN {X 0,Y 176.301,Z 388.064,A -85,B 0,C 180,E1 -22776.869,E2 -22776.869} C_VEL
LIN {X 0,Y 176.693,Z 385.928,A -85,B 0,C 180,E1 -22780.004,E2 -22780.004} C_VEL
LIN {X 0,Y 176.467,Z 384.366,A -85,B 0,C 180,E1 -22781.842,E2 -22781.842} C_VEL
LIN {X 0,Y 174.669,Z 381.212,A -85,B 0,C 180,E1 -22784.852,E2 -22784.852} C_VEL
LIN {X 0,Y 173.228,Z 377.436,A -85,B 0,C 180,E1 -22787.842,E2 -22787.842} C_VEL
LIN {X 0,Y 173.564,Z 374.792,A -85,B 0,C 180,E1 -22789.596,E2 -22789.596} C_VEL
LIN {X 0,Y 176.105,Z 368.669,A -85,B 0,C 180,E1 -22792.899,E2 -22792.899} C_VEL
LIN {X 0,Y 179.074,Z 360.892,A -85,B 0,C 180,E1 -22796.202,E2 -22796.202} C_VEL
LIN {X 0,Y 182.83,Z 351.166,A -85,B 0,C 180,E1 -22799.349,E2 -22799.349} C_VEL
LIN {X 0,Y 184.368,Z 342.101,A -85,B 0,C 180,E1 -22801.932,E2 -22801.932} C_VEL
LIN {X 0,Y 185.101,Z 332.02,A -85,B 0,C 180,E1 -22804.453,E2 -22804.453} C_VEL
LIN {X 0,Y 185.029,Z 321.592,A -85,B 0,C 180,E1 -22806.766,E2 -22806.766} C_VEL
LIN {X 0,Y 184.151,Z 310.902,A -85,B 0,C 180,E1 -22808.91,E2 -22808.91} C_VEL
LIN {X 0,Y 182.279,Z 300.165,A -85,B 0,C 180,E1 -22810.955,E2 -22810.955} C_VEL
LIN {X 0,Y 179.952,Z 293.536,A -85,B 0,C 180,E1 -22812.389,E2 -22812.389} C_VEL
LIN {X 0,Y 178.232,Z 289.887,A -85,B 0,C 180,E1 -22813.262,E2 -22813.262} C_VEL
LIN {X 0,Y 176.273,Z 285.781,A -85,B 0,C 180,E1 -22814.241,E2 -22814.241} C_VEL
LIN {X 0,Y 174.466,Z 282.783,A -85,B 0,C 180,E1 -22815.072,E2 -22815.072} C_VEL
LIN {X 0,Y 173.875,Z 280.717,A -85,B 0,C 180,E1 -22815.49,E2 -22815.49} C_VEL
LIN {X 0,Y 173.141,Z 277.325,A -85,B 0,C 180,E1 -22820.466,E2 -22820.466} C_VEL
LIN {X 0,Y 172.687,Z 274.359,A -85,B 0,C 180,E1 -22825.266,E2 -22825.266} C_VEL
LIN {X 0,Y 172.142,Z 271.317,A -85,B 0,C 180,E1 -22830.665,E2 -22830.665} C_VEL
LIN {X 0,Y 171.742,Z 268.76,A -85,B 0,C 180,E1 -22835.844,E2 -22835.844} C_VEL
LIN {X 0,Y 171.534,Z 267.12,A -85,B 0,C 180,E1 -22840.133,E2 -22840.133} C_VEL
LIN {X 0,Y 171.556,Z 267.116,A -85,B 0,C 180,E1 -22843.336,E2 -22843.336} C_VEL
LIN {X 0,Y 171.771,Z 267.089,A -85,B 0,C 180,E1 -22849.103,E2 -22849.103} C_VEL
LIN {X 0,Y 171.873,Z 267.074,A -85,B 0,C 180,E1 -22852.954,E2 -22852.954} C_VEL
LIN {X 0,Y 172.102,Z 267.046,A -85,B 0,C 180,E1 -22857.66,E2 -22857.66} C_VEL
LIN {X 0,Y 172.314,Z 267.019,A -85,B 0,C 180,E1 -22860,E2 -22860} C_VEL
LIN {X 0,Y 171.799,Z 267.085,A -85,B 0,C 180,E1 -22864.693,E2 -22864.693} C_VEL
LIN {X 0,Y 171.85,Z 267.077,A -85,B 0,C 180,E1 -22869.415,E2 -22869.415} C_VEL
LIN {X 0,Y 171.562,Z 267.114,A -85,B 0,C 180,E1 -22874.229,E2 -22874.229} C_VEL
LIN {X 0,Y 171.518,Z 267.12,A -85,B 0,C 180,E1 -22879.534,E2 -22879.534} C_VEL
LIN {X 0,Y 171.446,Z 267.128,A -85,B 0,C 180,E1 -22885.598,E2 -22885.598} C_VEL
LIN {X 0,Y 171.42,Z 267.131,A -85,B 0,C 180,E1 -22890.573,E2 -22890.573} C_VEL
LIN {X 0,Y 171.395,Z 267.132,A -85,B 0,C 180,E1 -22895.035,E2 -22895.035} C_VEL
LIN {X 0,Y 171.361,Z 267.136,A -85,B 0,C 180,E1 -22898.807,E2 -22898.807} C_VEL
LIN {X 0,Y 171.331,Z 267.264,A -85,B 0,C 180,E1 -22903.836,E2 -22903.836} C_VEL
LIN {X 0,Y 172.305,Z 269.942,A -85,B 0,C 180,E1 -22904.421,E2 -22904.421} C_VEL
LIN {X 0,Y 174.339,Z 272.329,A -85,B 0,C 180,E1 -22905.331,E2 -22905.331} C_VEL
LIN {X 0,Y 176.46,Z 275.978,A -85,B 0,C 180,E1 -22906.417,E2 -22906.417} C_VEL
LIN {X 0,Y 181.337,Z 285.425,A -85,B 0,C 180,E1 -22909.09,E2 -22909.09} C_VEL
LIN {X 0,Y 184.962,Z 294.935,A -85,B 0,C 180,E1 -22911.584,E2 -22911.584} C_VEL
LIN {X 0,Y 187.493,Z 304.994,A -85,B 0,C 180,E1 -22914.153,E2 -22914.153} C_VEL
LIN {X 0,Y 188.942,Z 314.686,A -85,B 0,C 180,E1 -22916.729,E2 -22916.729} C_VEL
LIN {X 0,Y 189.204,Z 320.585,A -85,B 0,C 180,E1 -22918.354,E2 -22918.354} C_VEL
LIN {X 0,Y 186.251,Z 329.846,A -85,B 0,C 180,E1 -22920.623,E2 -22920.623} C_VEL
LIN {X 0,Y 183.086,Z 338.288,A -85,B 0,C 180,E1 -22923.189,E2 -22923.189} C_VEL
LIN {X 0,Y 179.682,Z 346.494,A -85,B 0,C 180,E1 -22926.364,E2 -22926.364} C_VEL
LIN {X 0,Y 177.22,Z 352.102,A -85,B 0,C 180,E1 -22929.089,E2 -22929.089} C_VEL
LIN {X 0,Y 174.714,Z 357.564,A -85,B 0,C 180,E1 -22932.44,E2 -22932.44} C_VEL
LIN {X 0,Y 172.701,Z 361.847,A -85,B 0,C 180,E1 -22935.867,E2 -22935.867} C_VEL
LIN {X 0,Y 171.73,Z 364.106,A -85,B 0,C 180,E1 -22938.192,E2 -22938.192} C_VEL
LIN {X 0,Y 170.96,Z 365.994,A -85,B 0,C 180,E1 -22940.618,E2 -22940.618} C_VEL
LIN {X 0,Y 169.94,Z 368.297,A -85,B 0,C 180,E1 -22945.255,E2 -22945.255} C_VEL
LIN {X 0,Y 169.529,Z 369.129,A -85,B 0,C 180,E1 -22950,E2 -22950} C_VEL
LIN {X 0,Y 169.93,Z 368.348,A -85,B 0,C 180,E1 -22954.744,E2 -22954.744} C_VEL
LIN {X 0,Y 170.699,Z 366.43,A -85,B 0,C 180,E1 -22958.836,E2 -22958.836} C_VEL
LIN {X 0,Y 172.167,Z 363.197,A -85,B 0,C 180,E1 -22962.974,E2 -22962.974} C_VEL
LIN {X 0,Y 173.915,Z 359.332,A -85,B 0,C 180,E1 -22966.432,E2 -22966.432} C_VEL
LIN {X 0,Y 176.252,Z 354.335,A -85,B 0,C 180,E1 -22969.812,E2 -22969.812} C_VEL
LIN {X 0,Y 179.062,Z 348.037,A -85,B 0,C 180,E1 -22973.109,E2 -22973.109} C_VEL
LIN {X 0,Y 182.424,Z 340.148,A -85,B 0,C 180,E1 -22976.298,E2 -22976.298} C_VEL
LIN {X 0,Y 185.567,Z 332.101,A -85,B 0,C 180,E1 -22978.874,E2 -22978.874} C_VEL
LIN {X 0,Y 188.782,Z 322.291,A -85,B 0,C 180,E1 -22981.412,E2 -22981.412} C_VEL
LIN {X 0,Y 189.409,Z 320.031,A -85,B 0,C 180,E1 -22981.92,E2 -22981.92} C_VEL
LIN {X 0,Y 188.523,Z 310.774,A -85,B 0,C 180,E1 -22984.485,E2 -22984.485} C_VEL
LIN {X 0,Y 187.005,Z 302.565,A -85,B 0,C 180,E1 -22986.645,E2 -22986.645} C_VEL
LIN {X 0,Y 184.581,Z 293.679,A -85,B 0,C 180,E1 -22988.919,E2 -22988.919} C_VEL
LIN {X 0,Y 181.009,Z 284.629,A -85,B 0,C 180,E1 -22991.304,E2 -22991.304} C_VEL
LIN {X 0,Y 176.185,Z 275.631,A -85,B 0,C 180,E1 -22993.903,E2 -22993.903} C_VEL
LIN {X 0,Y 174.298,Z 272.241,A -85,B 0,C 180,E1 -22994.888,E2 -22994.888} C_VEL
LIN {X 0,Y 172.023,Z 269.476,A -85,B 0,C 180,E1 -22995.922,E2 -22995.922} C_VEL
LIN {X 0,Y 171.304,Z 267.141,A -85,B 0,C 180,E1 -22996.407,E2 -22996.407} C_VEL
LIN {X 0,Y 171.388,Z 267.136,A -85,B 0,C 180,E1 -23002.041,E2 -23002.041} C_VEL
LIN {X 0,Y 171.399,Z 267.135,A -85,B 0,C 180,E1 -23005.092,E2 -23005.092} C_VEL
LIN {X 0,Y 171.41,Z 267.134,A -85,B 0,C 180,E1 -23010.527,E2 -23010.527} C_VEL
LIN {X 0,Y 171.442,Z 267.129,A -85,B 0,C 180,E1 -23015.799,E2 -23015.799} C_VEL
LIN {X 0,Y 171.547,Z 267.114,A -85,B 0,C 180,E1 -23020.868,E2 -23020.868} C_VEL
LIN {X 0,Y 171.565,Z 267.11,A -85,B 0,C 180,E1 -23025.772,E2 -23025.772} C_VEL
LIN {X 0,Y 171.905,Z 267.072,A -85,B 0,C 180,E1 -23030.588,E2 -23030.588} C_VEL
LIN {X 0,Y 171.81,Z 267.082,A -85,B 0,C 180,E1 -23035.307,E2 -23035.307} C_VEL
LIN {X 0,Y 172.313,Z 267.017,A -85,B 0,C 180,E1 -23040,E2 -23040} C_VEL
LIN {X 0,Y 171.816,Z 267.084,A -85,B 0,C 180,E1 -23044.692,E2 -23044.692} C_VEL
LIN {X 0,Y 171.848,Z 267.075,A -85,B 0,C 180,E1 -23049.415,E2 -23049.415} C_VEL
LIN {X 0,Y 171.577,Z 267.112,A -85,B 0,C 180,E1 -23054.227,E2 -23054.227} C_VEL
LIN {X 0,Y 171.539,Z 267.116,A -85,B 0,C 180,E1 -23059.556,E2 -23059.556} C_VEL
LIN {X 0,Y 171.574,Z 267.713,A -85,B 0,C 180,E1 -23061.633,E2 -23061.633} C_VEL
LIN {X 0,Y 171.922,Z 270.071,A -85,B 0,C 180,E1 -23066.722,E2 -23066.722} C_VEL
LIN {X 0,Y 172.342,Z 272.861,A -85,B 0,C 180,E1 -23072.014,E2 -23072.014} C_VEL
LIN {X 0,Y 172.703,Z 274.91,A -85,B 0,C 180,E1 -23075.523,E2 -23075.523} C_VEL
LIN {X 0,Y 173.307,Z 278.02,A -85,B 0,C 180,E1 -23080.454,E2 -23080.454} C_VEL
LIN {X 0,Y 173.905,Z 280.817,A -85,B 0,C 180,E1 -23084.5,E2 -23084.5} C_VEL
LIN {X 0,Y 174.946,Z 283.809,A -85,B 0,C 180,E1 -23085.076,E2 -23085.076} C_VEL
LIN {X 0,Y 176.851,Z 286.863,A -85,B 0,C 180,E1 -23085.938,E2 -23085.938} C_VEL
LIN {X 0,Y 178.864,Z 290.964,A -85,B 0,C 180,E1 -23086.946,E2 -23086.946} C_VEL
LIN {X 0,Y 181.886,Z 298.538,A -85,B 0,C 180,E1 -23088.653,E2 -23088.653} C_VEL
LIN {X 0,Y 183.85,Z 308.586,A -85,B 0,C 180,E1 -23090.578,E2 -23090.578} C_VEL
LIN {X 0,Y 185.027,Z 320.284,A -85,B 0,C 180,E1 -23092.907,E2 -23092.907} C_VEL
LIN {X 0,Y 185.169,Z 331.222,A -85,B 0,C 180,E1 -23095.297,E2 -23095.297} C_VEL
LIN {X 0,Y 184.522,Z 341.233,A -85,B 0,C 180,E1 -23097.776,E2 -23097.776} C_VEL
LIN {X 0,Y 183.33,Z 349.534,A -85,B 0,C 180,E1 -23100.109,E2 -23100.109} C_VEL
LIN {X 0,Y 180.872,Z 356.46,A -85,B 0,C 180,E1 -23102.207,E2 -23102.207} C_VEL
LIN {X 0,Y 177.922,Z 363.928,A -85,B 0,C 180,E1 -23104.935,E2 -23104.935} C_VEL
LIN {X 0,Y 175.234,Z 371.037,A -85,B 0,C 180,E1 -23108.224,E2 -23108.224} C_VEL
LIN {X 0,Y 173.192,Z 375.926,A -85,B 0,C 180,E1 -23111.057,E2 -23111.057} C_VEL
LIN {X 0,Y 171.218,Z 380.684,A -85,B 0,C 180,E1 -23114.526,E2 -23114.526} C_VEL
LIN {X 0,Y 170.039,Z 384.342,A -85,B 0,C 180,E1 -23118.074,E2 -23118.074} C_VEL
LIN {X 0,Y 169.518,Z 386.234,A -85,B 0,C 180,E1 -23120.455,E2 -23120.455} C_VEL
LIN {X 0,Y 169.243,Z 387.66,A -85,B 0,C 180,E1 -23122.844,E2 -23122.844} C_VEL
LIN {X 0,Y 169.173,Z 388.81,A -85,B 0,C 180,E1 -23125.591,E2 -23125.591} C_VEL
LIN {X 0,Y 169.385,Z 389.542,A -85,B 0,C 180,E1 -23130,E2 -23130} C_VEL
LIN {X 0,Y 169.164,Z 388.805,A -85,B 0,C 180,E1 -23134.369,E2 -23134.369} C_VEL
LIN {X 0,Y 169.239,Z 387.635,A -85,B 0,C 180,E1 -23137.157,E2 -23137.157} C_VEL
LIN {X 0,Y 169.616,Z 385.73,A -85,B 0,C 180,E1 -23140.132,E2 -23140.132} C_VEL
LIN {X 0,Y 170.737,Z 381.948,A -85,B 0,C 180,E1 -23144.299,E2 -23144.299} C_VEL
LIN {X 0,Y 172.453,Z 377.55,A -85,B 0,C 180,E1 -23147.798,E2 -23147.798} C_VEL
LIN {X 0,Y 173.564,Z 374.792,A -85,B 0,C 180,E1 -23149.596,E2 -23149.596} C_VEL
LIN {X 0,Y 174.01,Z 371.967,A -85,B 0,C 180,E1 -23151.304,E2 -23151.304} C_VEL
LIN {X 0,Y 173.294,Z 366.914,A -85,B 0,C 180,E1 -23154.115,E2 -23154.115} C_VEL
LIN {X 0,Y 172.929,Z 361.342,A -85,B 0,C 180,E1 -23156.818,E2 -23156.818} C_VEL
LIN {X 0,Y 173.896,Z 357.578,A -85,B 0,C 180,E1 -23158.302,E2 -23158.302} C_VEL
LIN {X 0,Y 176.535,Z 350.725,A -85,B 0,C 180,E1 -23160.504,E2 -23160.504} C_VEL
LIN {X 0,Y 178.06,Z 341.646,A -85,B 0,C 180,E1 -23163.206,E2 -23163.206} C_VEL
LIN {X 0,Y 178.783,Z 332.958,A -85,B 0,C 180,E1 -23165.487,E2 -23165.487} C_VEL
LIN {X 0,Y 178.839,Z 321.444,A -85,B 0,C 180,E1 -23168.191,E2 -23168.191} C_VEL
LIN {X 0,Y 178.084,Z 311.438,A -85,B 0,C 180,E1 -23170.319,E2 -23170.319} C_VEL
LIN {X 0,Y 176.721,Z 303.05,A -85,B 0,C 180,E1 -23172.053,E2 -23172.053} C_VEL
LIN {X 0,Y 174.795,Z 297.277,A -85,B 0,C 180,E1 -23173.422,E2 -23173.422} C_VEL
LIN {X 0,Y 171.615,Z 290.349,A -85,B 0,C 180,E1 -23175.262,E2 -23175.262} C_VEL
LIN {X 0,Y 169.618,Z 286.281,A -85,B 0,C 180,E1 -23176.371,E2 -23176.371} C_VEL
LIN {X 0,Y 166.959,Z 281.909,A -85,B 0,C 180,E1 -23177.736,E2 -23177.736} C_VEL
LIN {X 0,Y 166.451,Z 280.103,A -85,B 0,C 180,E1 -23178.094,E2 -23178.094} C_VEL
LIN {X 0,Y 165.808,Z 276.684,A -85,B 0,C 180,E1 -23183.644,E2 -23183.644} C_VEL
LIN {X 0,Y 165.322,Z 273.53,A -85,B 0,C 180,E1 -23189.327,E2 -23189.327} C_VEL
LIN {X 0,Y 164.898,Z 270.833,A -85,B 0,C 180,E1 -23194.773,E2 -23194.773} C_VEL
LIN {X 0,Y 164.588,Z 268.62,A -85,B 0,C 180,E1 -23200.025,E2 -23200.025} C_VEL
LIN {X 0,Y 164.486,Z 267.998,A -85,B 0,C 180,E1 -23202.597,E2 -23202.597} C_VEL
LIN {X 0,Y 164.706,Z 267.969,A -85,B 0,C 180,E1 -23208.939,E2 -23208.939} C_VEL
LIN {X 0,Y 164.833,Z 267.951,A -85,B 0,C 180,E1 -23212.651,E2 -23212.651} C_VEL
LIN {X 0,Y 165.051,Z 267.925,A -85,B 0,C 180,E1 -23217.56,E2 -23217.56} C_VEL
LIN {X 0,Y 165.278,Z 267.896,A -85,B 0,C 180,E1 -23220,E2 -23220} C_VEL
LIN {X 0,Y 164.749,Z 267.964,A -85,B 0,C 180,E1 -23224.894,E2 -23224.894} C_VEL
LIN {X 0,Y 164.83,Z 267.954,A -85,B 0,C 180,E1 -23227.349,E2 -23227.349} C_VEL
LIN {X 0,Y 164.705,Z 267.968,A -85,B 0,C 180,E1 -23231.061,E2 -23231.061} C_VEL
LIN {X 0,Y 164.455,Z 267.997,A -85,B 0,C 180,E1 -23237.406,E2 -23237.406} C_VEL
LIN {X 0,Y 164.452,Z 267.999,A -85,B 0,C 180,E1 -23239.992,E2 -23239.992} C_VEL
LIN {X 0,Y 164.373,Z 268.008,A -85,B 0,C 180,E1 -23246.117,E2 -23246.117} C_VEL
LIN {X 0,Y 164.36,Z 268.01,A -85,B 0,C 180,E1 -23251.217,E2 -23251.217} C_VEL
LIN {X 0,Y 164.297,Z 268.014,A -85,B 0,C 180,E1 -23256.789,E2 -23256.789} C_VEL
LIN {X 0,Y 164.293,Z 268.043,A -85,B 0,C 180,E1 -23261.227,E2 -23261.227} C_VEL
LIN {X 0,Y 165.206,Z 270.738,A -85,B 0,C 180,E1 -23261.864,E2 -23261.864} C_VEL
LIN {X 0,Y 167.451,Z 273.39,A -85,B 0,C 180,E1 -23262.998,E2 -23262.998} C_VEL
LIN {X 0,Y 169.318,Z 276.58,A -85,B 0,C 180,E1 -23264.068,E2 -23264.068} C_VEL
LIN {X 0,Y 170.644,Z 278.629,A -85,B 0,C 180,E1 -23264.781,E2 -23264.781} C_VEL
LIN {X 0,Y 174.729,Z 286.249,A -85,B 0,C 180,E1 -23267.228,E2 -23267.228} C_VEL
LIN {X 0,Y 178.293,Z 294.953,A -85,B 0,C 180,E1 -23269.766,E2 -23269.766} C_VEL
LIN {X 0,Y 180.418,Z 302.504,A -85,B 0,C 180,E1 -23271.848,E2 -23271.848} C_VEL
LIN {X 0,Y 182.018,Z 310.876,A -85,B 0,C 180,E1 -23274.179,E2 -23274.179} C_VEL
LIN {X 0,Y 182.935,Z 320.136,A -85,B 0,C 180,E1 -23276.876,E2 -23276.876} C_VEL
LIN {X 0,Y 182.84,Z 322.162,A -85,B 0,C 180,E1 -23277.443,E2 -23277.443} C_VEL
LIN {X 0,Y 179.435,Z 332.07,A -85,B 0,C 180,E1 -23280.04,E2 -23280.04} C_VEL
LIN {X 0,Y 175.529,Z 341.664,A -85,B 0,C 180,E1 -23283.228,E2 -23283.228} C_VEL
LIN {X 0,Y 172.16,Z 349.301,A -85,B 0,C 180,E1 -23286.545,E2 -23286.545} C_VEL
LIN {X 0,Y 168.81,Z 356.312,A -85,B 0,C 180,E1 -23290.545,E2 -23290.545} C_VEL
LIN {X 0,Y 166.5,Z 360.975,A -85,B 0,C 180,E1 -23294.075,E2 -23294.075} C_VEL
LIN {X 0,Y 164.809,Z 364.533,A -85,B 0,C 180,E1 -23297.689,E2 -23297.689} C_VEL
LIN {X 0,Y 163.855,Z 366.639,A -85,B 0,C 180,E1 -23300.578,E2 -23300.578} C_VEL
LIN {X 0,Y 162.881,Z 368.724,A -85,B 0,C 180,E1 -23305.049,E2 -23305.049} C_VEL
LIN {X 0,Y 162.467,Z 369.555,A -85,B 0,C 180,E1 -23310,E2 -23310} C_VEL
LIN {X 0,Y 162.566,Z 369.359,A -85,B 0,C 180,E1 -23312.477,E2 -23312.477} C_VEL
LIN {X 0,Y 162.87,Z 368.774,A -85,B 0,C 180,E1 -23314.951,E2 -23314.951} C_VEL
LIN {X 0,Y 163.91,Z 366.47,A -85,B 0,C 180,E1 -23319.875,E2 -23319.875} C_VEL
LIN {X 0,Y 165.265,Z 363.623,A -85,B 0,C 180,E1 -23323.526,E2 -23323.526} C_VEL
LIN {X 0,Y 167.136,Z 359.757,A -85,B 0,C 180,E1 -23327.118,E2 -23327.118} C_VEL
LIN {X 0,Y 169.614,Z 354.759,A -85,B 0,C 180,E1 -23330.622,E2 -23330.622} C_VEL
LIN {X 0,Y 172.559,Z 348.462,A -85,B 0,C 180,E1 -23334.034,E2 -23334.034} C_VEL
LIN {X 0,Y 176.105,Z 340.572,A -85,B 0,C 180,E1 -23337.319,E2 -23337.319} C_VEL
LIN {X 0,Y 179.399,Z 332.524,A -85,B 0,C 180,E1 -23339.966,E2 -23339.966} C_VEL
LIN {X 0,Y 182.784,Z 322.713,A -85,B 0,C 180,E1 -23342.568,E2 -23342.568} C_VEL
LIN {X 0,Y 183.033,Z 320.649,A -85,B 0,C 180,E1 -23343.124,E2 -23343.124} C_VEL
LIN {X 0,Y 182.281,Z 312.25,A -85,B 0,C 180,E1 -23345.594,E2 -23345.594} C_VEL
LIN {X 0,Y 180.731,Z 303.45,A -85,B 0,C 180,E1 -23348.053,E2 -23348.053} C_VEL
LIN {X 0,Y 178.411,Z 295.164,A -85,B 0,C 180,E1 -23350.345,E2 -23350.345} C_VEL
LIN {X 0,Y 175.614,Z 288.085,A -85,B 0,C 180,E1 -23352.408,E2 -23352.408} C_VEL
LIN {X 0,Y 171.5,Z 280.162,A -85,B 0,C 180,E1 -23354.913,E2 -23354.913} C_VEL
LIN {X 0,Y 169.563,Z 276.895,A -85,B 0,C 180,E1 -23356.013,E2 -23356.013} C_VEL
LIN {X 0,Y 167.477,Z 273.485,A -85,B 0,C 180,E1 -23357.192,E2 -23357.192} C_VEL
LIN {X 0,Y 166.944,Z 272.692,A -85,B 0,C 180,E1 -23357.476,E2 -23357.476} C_VEL
LIN {X 0,Y 165.108,Z 270.531,A -85,B 0,C 180,E1 -23358.412,E2 -23358.412} C_VEL
LIN {X 0,Y 164.304,Z 268.018,A -85,B 0,C 180,E1 -23359.031,E2 -23359.031} C_VEL
LIN {X 0,Y 164.331,Z 268.016,A -85,B 0,C 180,E1 -23364.349,E2 -23364.349} C_VEL
LIN {X 0,Y 164.371,Z 268.007,A -85,B 0,C 180,E1 -23369.13,E2 -23369.13} C_VEL
LIN {X 0,Y 164.396,Z 268.003,A -85,B 0,C 180,E1 -23374.69,E2 -23374.69} C_VEL
LIN {X 0,Y 164.441,Z 268.002,A -85,B 0,C 180,E1 -23380.094,E2 -23380.094} C_VEL
LIN {X 0,Y 164.492,Z 267.99,A -85,B 0,C 180,E1 -23385.146,E2 -23385.146} C_VEL
LIN {X 0,Y 164.834,Z 267.951,A -85,B 0,C 180,E1 -23390.18,E2 -23390.18} C_VEL
LIN {X 0,Y 164.861,Z 267.944,A -85,B 0,C 180,E1 -23392.652,E2 -23392.652} C_VEL
LIN {X 0,Y 165.277,Z 267.893,A -85,B 0,C 180,E1 -23400,E2 -23400} C_VEL
LIN {X 0,Y 164.765,Z 267.963,A -85,B 0,C 180,E1 -23404.894,E2 -23404.894} C_VEL
LIN {X 0,Y 164.831,Z 267.951,A -85,B 0,C 180,E1 -23407.349,E2 -23407.349} C_VEL
LIN {X 0,Y 164.704,Z 267.97,A -85,B 0,C 180,E1 -23411.061,E2 -23411.061} C_VEL
LIN {X 0,Y 164.484,Z 267.994,A -85,B 0,C 180,E1 -23417.403,E2 -23417.403} C_VEL
LIN {X 0,Y 164.609,Z 268.717,A -85,B 0,C 180,E1 -23420.067,E2 -23420.067} C_VEL
LIN {X 0,Y 165.003,Z 271.546,A -85,B 0,C 180,E1 -23426.561,E2 -23426.561} C_VEL
LIN {X 0,Y 165.39,Z 274.199,A -85,B 0,C 180,E1 -23431.802,E2 -23431.802} C_VEL
LIN {X 0,Y 165.807,Z 276.807,A -85,B 0,C 180,E1 -23436.4,E2 -23436.4} C_VEL
LIN {X 0,Y 166.474,Z 280.169,A -85,B 0,C 180,E1 -23441.831,E2 -23441.831} C_VEL
LIN {X 0,Y 167.63,Z 283.327,A -85,B 0,C 180,E1 -23442.537,E2 -23442.537} C_VEL
LIN {X 0,Y 169.754,Z 286.579,A -85,B 0,C 180,E1 -23443.599,E2 -23443.599} C_VEL
LIN {X 0,Y 171.864,Z 290.699,A -85,B 0,C 180,E1 -23444.759,E2 -23444.759} C_VEL
LIN {X 0,Y 175.644,Z 299.215,A -85,B 0,C 180,E1 -23446.989,E2 -23446.989} C_VEL
LIN {X 0,Y 177.245,Z 305.312,A -85,B 0,C 180,E1 -23448.346,E2 -23448.346} C_VEL
LIN {X 0,Y 178.549,Z 315.994,A -85,B 0,C 180,E1 -23450.554,E2 -23450.554} C_VEL
LIN {X 0,Y 179.019,Z 325.908,A -85,B 0,C 180,E1 -23452.758,E2 -23452.758} C_VEL
